	(*-------------------------------------------------------------------------------- Robot Tool Changer Faults -------------------------------------------------------------------*)
	(*Fault1301 - R1 Tool Changer Fault*)
		Fault_Tmrs[1301].PT:= Short_Faults;
		Fault_Tmrs[1301]();
		Fault_Tmrs[1301].IN:= (GTAC_CONFIG.Option_Robot_Count>=1) AND
							MAIN.R1.ToolChanger_FLT;
		Out_To_ICxx.System_Faults[1301]:=Fault_Tmrs[1301].Q;
	(*Fault1302 - R2 Tool Changer Fault*)
		Fault_Tmrs[1302].PT:= Short_Faults;
		Fault_Tmrs[1302]();
		Fault_Tmrs[1302].IN:= (GTAC_CONFIG.Option_Robot_Count>=2) AND
							MAIN.R2.ToolChanger_FLT;
		Out_To_ICxx.System_Faults[1302]:=Fault_Tmrs[1302].Q;
	(*Fault1303 - R3 Tool Changer Fault*)
		Fault_Tmrs[1303].PT:= Short_Faults;
		Fault_Tmrs[1303]();
		Fault_Tmrs[1303].IN:= (GTAC_CONFIG.Option_Robot_Count>=3) AND
							MAIN.R3.ToolChanger_FLT;
		Out_To_ICxx.System_Faults[1303]:=Fault_Tmrs[1303].Q;
	(*Fault1304 - R4 Tool Changer Fault*)
		Fault_Tmrs[1304].PT:= Short_Faults;
		Fault_Tmrs[1304]();
		Fault_Tmrs[1304].IN:= (GTAC_CONFIG.Option_Robot_Count>=4) AND
							MAIN.R4.ToolChanger_FLT;
		Out_To_ICxx.System_Faults[1304]:=Fault_Tmrs[1304].Q;
	(*Fault1305 - R5 Tool Changer Fault*)
		Fault_Tmrs[1305].PT:= Short_Faults;
		Fault_Tmrs[1305]();
		Fault_Tmrs[1305].IN:= (GTAC_CONFIG.Option_Robot_Count>=5) AND
							MAIN.R5.ToolChanger_FLT;
		Out_To_ICxx.System_Faults[1305]:=Fault_Tmrs[1305].Q;
	(*Fault1306 - R6 Tool Changer Fault*)
		Fault_Tmrs[1306].PT:= Short_Faults;
		Fault_Tmrs[1306]();
		Fault_Tmrs[1306].IN:= (GTAC_CONFIG.Option_Robot_Count>=6) AND
							MAIN.R6.ToolChanger_FLT;
		Out_To_ICxx.System_Faults[1306]:=Fault_Tmrs[1306].Q;
	(*Fault1307 - R7 Tool Changer Fault*)
		Fault_Tmrs[1307].PT:= Short_Faults;
		Fault_Tmrs[1307]();
		Fault_Tmrs[1307].IN:= (GTAC_CONFIG.Option_Robot_Count>=7) AND
							MAIN.R7.ToolChanger_FLT;
		Out_To_ICxx.System_Faults[1307]:=Fault_Tmrs[1307].Q;
	(*Fault1308 - R8 Tool Changer Fault*)
		Fault_Tmrs[1308].PT:= Short_Faults;
		Fault_Tmrs[1308]();
		Fault_Tmrs[1308].IN:= (GTAC_CONFIG.Option_Robot_Count>=8) AND
							MAIN.R8.ToolChanger_FLT;
		Out_To_ICxx.System_Faults[1308]:=Fault_Tmrs[1308].Q;
	(*Fault1309 - R9 Tool Changer Fault*)
		Fault_Tmrs[1309].PT:= Short_Faults;
		Fault_Tmrs[1309]();
		Fault_Tmrs[1309].IN:= (GTAC_CONFIG.Option_Robot_Count>=9) AND
							MAIN.R9.ToolChanger_FLT;
		Out_To_ICxx.System_Faults[1309]:=Fault_Tmrs[1309].Q;
	(*Fault1310 - R10 Tool Changer Fault*)
		Fault_Tmrs[1310].PT:= Short_Faults;
		Fault_Tmrs[1310]();
		Fault_Tmrs[1310].IN:= (GTAC_CONFIG.Option_Robot_Count>=10) AND
							MAIN.R10.ToolChanger_FLT;
		Out_To_ICxx.System_Faults[1310]:=Fault_Tmrs[1310].Q;
	(*Fault1311 - R11 Tool Changer Fault*)
		Fault_Tmrs[1311].PT:= Short_Faults;
		Fault_Tmrs[1311]();
		Fault_Tmrs[1311].IN:= (GTAC_CONFIG.Option_Robot_Count>=11) AND
							MAIN.R11.ToolChanger_FLT;
		Out_To_ICxx.System_Faults[1311]:=Fault_Tmrs[1311].Q;
	(*Fault1312 - R12 Tool Changer Fault*)
		Fault_Tmrs[1312].PT:= Short_Faults;
		Fault_Tmrs[1312]();
		Fault_Tmrs[1312].IN:= (GTAC_CONFIG.Option_Robot_Count>=12) AND
							MAIN.R12.ToolChanger_FLT;
		Out_To_ICxx.System_Faults[1312]:=Fault_Tmrs[1312].Q;
	(*Fault1313 - R13 Tool Changer Fault*)
		Fault_Tmrs[1313].PT:= Short_Faults;
		Fault_Tmrs[1313]();
		Fault_Tmrs[1313].IN:= (GTAC_CONFIG.Option_Robot_Count>=13) AND
							MAIN.R13.ToolChanger_FLT;
		Out_To_ICxx.System_Faults[1313]:=Fault_Tmrs[1313].Q;
	(*Fault1314 - R14 Tool Changer Fault*)
		Fault_Tmrs[1314].PT:= Short_Faults;
		Fault_Tmrs[1314]();
		Fault_Tmrs[1314].IN:= (GTAC_CONFIG.Option_Robot_Count>=14) AND
							MAIN.R14.ToolChanger_FLT;
		Out_To_ICxx.System_Faults[1314]:=Fault_Tmrs[1314].Q;
	(*Fault1315 - R15 Tool Changer Fault*)
		Fault_Tmrs[1315].PT:= Short_Faults;
		Fault_Tmrs[1315]();
		Fault_Tmrs[1315].IN:= (GTAC_CONFIG.Option_Robot_Count>=15) AND
							MAIN.R15.ToolChanger_FLT;
		Out_To_ICxx.System_Faults[1315]:=Fault_Tmrs[1315].Q;
	(*Fault1316 - R16 Tool Changer Fault*)
		Fault_Tmrs[1316].PT:= Short_Faults;
		Fault_Tmrs[1316]();
		Fault_Tmrs[1316].IN:= (GTAC_CONFIG.Option_Robot_Count>=16) AND
							MAIN.R16.ToolChanger_FLT;
		Out_To_ICxx.System_Faults[1316]:=Fault_Tmrs[1316].Q;
	(*Fault1317 - R17 Tool Changer Fault*)
		Fault_Tmrs[1317].PT:= Short_Faults;
		Fault_Tmrs[1317]();
		Fault_Tmrs[1317].IN:= (GTAC_CONFIG.Option_Robot_Count>=17) AND
							MAIN.R17.ToolChanger_FLT;
		Out_To_ICxx.System_Faults[1317]:=Fault_Tmrs[1317].Q;
	(*Fault1318 - R18 Tool Changer Fault*)
		Fault_Tmrs[1318].PT:= Short_Faults;
		Fault_Tmrs[1318]();
		Fault_Tmrs[1318].IN:= (GTAC_CONFIG.Option_Robot_Count>=18) AND
							MAIN.R18.ToolChanger_FLT;
		Out_To_ICxx.System_Faults[1318]:=Fault_Tmrs[1318].Q;
	(*Fault1319 - R19 Tool Changer Fault*)
		Fault_Tmrs[1319].PT:= Short_Faults;
		Fault_Tmrs[1319]();
		Fault_Tmrs[1319].IN:= (GTAC_CONFIG.Option_Robot_Count>=19) AND
							MAIN.R19.ToolChanger_FLT;
		Out_To_ICxx.System_Faults[1319]:=Fault_Tmrs[1319].Q;
	(*Fault1320 - R20 Tool Changer Fault*)
		Fault_Tmrs[1320].PT:= Short_Faults;
		Fault_Tmrs[1320]();
		Fault_Tmrs[1320].IN:= (GTAC_CONFIG.Option_Robot_Count>=20) AND
							MAIN.R20.ToolChanger_FLT;
		Out_To_ICxx.System_Faults[1320]:=Fault_Tmrs[1320].Q;
	(*Fault1321 - R21 Tool Changer Fault*)
		Fault_Tmrs[1321].PT:= Short_Faults;
		Fault_Tmrs[1321]();
		Fault_Tmrs[1321].IN:= (GTAC_CONFIG.Option_Robot_Count>=21) AND
							MAIN.R21.ToolChanger_FLT;
		Out_To_ICxx.System_Faults[1321]:=Fault_Tmrs[1321].Q;
	(*Fault1322 - R22 Tool Changer Fault*)
		Fault_Tmrs[1322].PT:= Short_Faults;
		Fault_Tmrs[1322]();
		Fault_Tmrs[1322].IN:= (GTAC_CONFIG.Option_Robot_Count>=22) AND
							MAIN.R22.ToolChanger_FLT;
		Out_To_ICxx.System_Faults[1322]:=Fault_Tmrs[1322].Q;
	(*Fault1323 - R23 Tool Changer Fault*)
		Fault_Tmrs[1323].PT:= Short_Faults;
		Fault_Tmrs[1323]();
		Fault_Tmrs[1323].IN:= (GTAC_CONFIG.Option_Robot_Count>=23) AND
							MAIN.R23.ToolChanger_FLT;
		Out_To_ICxx.System_Faults[1323]:=Fault_Tmrs[1323].Q;
	(*Fault1324 - R24 Tool Changer Fault*)
		Fault_Tmrs[1324].PT:= Short_Faults;
		Fault_Tmrs[1324]();
		Fault_Tmrs[1324].IN:= (GTAC_CONFIG.Option_Robot_Count>=24) AND
							MAIN.R24.ToolChanger_FLT;
		Out_To_ICxx.System_Faults[1324]:=Fault_Tmrs[1324].Q;
	(*Fault1325 - R25 Tool Changer Fault*)
		Fault_Tmrs[1325].PT:= Short_Faults;
		Fault_Tmrs[1325]();
		Fault_Tmrs[1325].IN:= (GTAC_CONFIG.Option_Robot_Count>=25) AND
							MAIN.R25.ToolChanger_FLT;
		Out_To_ICxx.System_Faults[1325]:=Fault_Tmrs[1325].Q;
	(*Fault1326 - R26 Tool Changer Fault*)
		Fault_Tmrs[1326].PT:= Short_Faults;
		Fault_Tmrs[1326]();
		Fault_Tmrs[1326].IN:= (GTAC_CONFIG.Option_Robot_Count>=26) AND
							MAIN.R26.ToolChanger_FLT;
		Out_To_ICxx.System_Faults[1326]:=Fault_Tmrs[1326].Q;
	(*Fault1327 - R27 Tool Changer Fault*)
		Fault_Tmrs[1327].PT:= Short_Faults;
		Fault_Tmrs[1327]();
		Fault_Tmrs[1327].IN:= (GTAC_CONFIG.Option_Robot_Count>=27) AND
							MAIN.R27.ToolChanger_FLT;
		Out_To_ICxx.System_Faults[1327]:=Fault_Tmrs[1327].Q;
	(*Fault1328 - R28 Tool Changer Fault*)
		Fault_Tmrs[1328].PT:= Short_Faults;
		Fault_Tmrs[1328]();
		Fault_Tmrs[1328].IN:= (GTAC_CONFIG.Option_Robot_Count>=28) AND
							MAIN.R28.ToolChanger_FLT;
		Out_To_ICxx.System_Faults[1328]:=Fault_Tmrs[1328].Q;
	(*Fault1329 - R29 Tool Changer Fault*)
		Fault_Tmrs[1329].PT:= Short_Faults;
		Fault_Tmrs[1329]();
		Fault_Tmrs[1329].IN:= (GTAC_CONFIG.Option_Robot_Count>=29) AND
							MAIN.R29.ToolChanger_FLT;
		Out_To_ICxx.System_Faults[1329]:=Fault_Tmrs[1329].Q;
	(*Fault1330 - R30 Tool Changer Fault*)
		Fault_Tmrs[1330].PT:= Short_Faults;
		Fault_Tmrs[1330]();
		Fault_Tmrs[1330].IN:= (GTAC_CONFIG.Option_Robot_Count>=30) AND
							MAIN.R30.ToolChanger_FLT;
		Out_To_ICxx.System_Faults[1330]:=Fault_Tmrs[1330].Q;

	(*-------------------------------------------------------------------------------- Robot EOAT Faults -------------------------------------------------------------------*)
	(*Fault1331 - EOAT01 Fault*)
		Fault_Tmrs[1331].PT:= Short_Faults;
		Fault_Tmrs[1331]();
		Fault_Tmrs[1331].IN:= (MAIN.R1.FB_In.Options.EOAT_Amount>=1) AND
							EOAT01.EOAT_FLT;
		Out_To_ICxx.System_Faults[1331]:=Fault_Tmrs[1331].Q;
	(*Fault1332 - EOAT02 Fault*)
		Fault_Tmrs[1332].PT:= Short_Faults;
		Fault_Tmrs[1332]();
		Fault_Tmrs[1332].IN:= (MAIN.R2.FB_In.Options.EOAT_Amount>=2) AND
							EOAT02.EOAT_FLT;
		Out_To_ICxx.System_Faults[1332]:=Fault_Tmrs[1332].Q;
	(*Fault1333 - EOAT03 Fault*)
		Fault_Tmrs[1333].PT:= Short_Faults;
		Fault_Tmrs[1333]();
		Fault_Tmrs[1333].IN:= (MAIN.R3.FB_In.Options.EOAT_Amount>=3) AND
							EOAT03.EOAT_FLT;
		Out_To_ICxx.System_Faults[1333]:=Fault_Tmrs[1333].Q;
	(*Fault1334 - EOAT04 Fault*)
		Fault_Tmrs[1334].PT:= Short_Faults;
		Fault_Tmrs[1334]();
		Fault_Tmrs[1334].IN:= (MAIN.R4.FB_In.Options.EOAT_Amount>=4) AND
							EOAT04.EOAT_FLT;
		Out_To_ICxx.System_Faults[1334]:=Fault_Tmrs[1334].Q;
	(*Fault1335 - EOAT05 Fault*)
		Fault_Tmrs[1335].PT:= Short_Faults;
		Fault_Tmrs[1335]();
		Fault_Tmrs[1335].IN:= (MAIN.R5.FB_In.Options.EOAT_Amount>=5) AND
							EOAT05.EOAT_FLT;
		Out_To_ICxx.System_Faults[1335]:=Fault_Tmrs[1335].Q;
	(*Fault1336 - EOAT06 Fault*)
		Fault_Tmrs[1336].PT:= Short_Faults;
		Fault_Tmrs[1336]();
		Fault_Tmrs[1336].IN:= (MAIN.R6.FB_In.Options.EOAT_Amount>=6) AND
							EOAT06.EOAT_FLT;
		Out_To_ICxx.System_Faults[1336]:=Fault_Tmrs[1336].Q;
	(*Fault1337 - EOAT07 Fault*)
		Fault_Tmrs[1337].PT:= Short_Faults;
		Fault_Tmrs[1337]();
		Fault_Tmrs[1337].IN:= (MAIN.R7.FB_In.Options.EOAT_Amount>=7) AND
							EOAT07.EOAT_FLT;
		Out_To_ICxx.System_Faults[1337]:=Fault_Tmrs[1337].Q;
	(*Fault1338 - EOAT08 Fault*)
		Fault_Tmrs[1338].PT:= Short_Faults;
		Fault_Tmrs[1338]();
		Fault_Tmrs[1338].IN:= (MAIN.R8.FB_In.Options.EOAT_Amount>=8) AND
							EOAT08.EOAT_FLT;
		Out_To_ICxx.System_Faults[1338]:=Fault_Tmrs[1338].Q;
	(*Fault1339 - EOAT09 Fault*)
		Fault_Tmrs[1339].PT:= Short_Faults;
		Fault_Tmrs[1339]();
		Fault_Tmrs[1339].IN:= (MAIN.R9.FB_In.Options.EOAT_Amount>=9) AND
							EOAT09.EOAT_FLT;
		Out_To_ICxx.System_Faults[1339]:=Fault_Tmrs[1339].Q;
	(*Fault1340 - EOAT10 Fault*)
		Fault_Tmrs[1340].PT:= Short_Faults;
		Fault_Tmrs[1340]();
		Fault_Tmrs[1340].IN:= (MAIN.R10.FB_In.Options.EOAT_Amount>=10) AND
							EOAT10.EOAT_FLT;
		Out_To_ICxx.System_Faults[1340]:=Fault_Tmrs[1340].Q;
(* Note  - add faults as more EOAT are added to the system.
	(*Fault1341 - EOAT11 Fault*)
		Fault_Tmrs[1341].PT:= Short_Faults;
		Fault_Tmrs[1341]();
		Fault_Tmrs[1341].IN:= (GTAC_CONFIG.Option_EOAT_Count>=11) AND
							EOAT11.EOAT_FLT;
		Out_To_ICxx.System_Faults[1341]:=Fault_Tmrs[1341].Q;
	(*Fault1342 - EOAT12 Fault*)
		Fault_Tmrs[1342].PT:= Short_Faults;
		Fault_Tmrs[1342]();
		Fault_Tmrs[1342].IN:= (GTAC_CONFIG.Option_EOAT_Count>=12) AND
							EOAT12.EOAT_FLT;
		Out_To_ICxx.System_Faults[1342]:=Fault_Tmrs[1342].Q;
	(*Fault1343 - EOAT13 Fault*)
		Fault_Tmrs[1343].PT:= Short_Faults;
		Fault_Tmrs[1343]();
		Fault_Tmrs[1343].IN:= (GTAC_CONFIG.Option_EOAT_Count>=13) AND
							EOAT13.EOAT_FLT;
		Out_To_ICxx.System_Faults[1343]:=Fault_Tmrs[1343].Q;
	(*Fault1344 - EOAT14 Fault*)
		Fault_Tmrs[1344].PT:= Short_Faults;
		Fault_Tmrs[1344]();
		Fault_Tmrs[1344].IN:= (GTAC_CONFIG.Option_EOAT_Count>=14) AND
							EOAT14.EOAT_FLT;
		Out_To_ICxx.System_Faults[1344]:=Fault_Tmrs[1344].Q;
	(*Fault1345 - EOAT15 Fault*)
		Fault_Tmrs[1345].PT:= Short_Faults;
		Fault_Tmrs[1345]();
		Fault_Tmrs[1345].IN:= (GTAC_CONFIG.Option_EOAT_Count>=15) AND
							EOAT15.EOAT_FLT;
		Out_To_ICxx.System_Faults[1345]:=Fault_Tmrs[1345].Q;
	(*Fault1346 - EOAT16 Fault*)
		Fault_Tmrs[1346].PT:= Short_Faults;
		Fault_Tmrs[1346]();
		Fault_Tmrs[1346].IN:= (GTAC_CONFIG.Option_EOAT_Count>=16) AND
							EOAT16.EOAT_FLT;
		Out_To_ICxx.System_Faults[1346]:=Fault_Tmrs[1346].Q;
	(*Fault1347 - EOAT17 Fault*)
		Fault_Tmrs[1347].PT:= Short_Faults;
		Fault_Tmrs[1347]();
		Fault_Tmrs[1347].IN:= (GTAC_CONFIG.Option_EOAT_Count>=17) AND
							EOAT17.EOAT_FLT;
		Out_To_ICxx.System_Faults[1347]:=Fault_Tmrs[1347].Q;
	(*Fault1348 - EOAT18 Fault*)
		Fault_Tmrs[1348].PT:= Short_Faults;
		Fault_Tmrs[1348]();
		Fault_Tmrs[1348].IN:= (GTAC_CONFIG.Option_EOAT_Count>=18) AND
							EOAT18.EOAT_FLT;
		Out_To_ICxx.System_Faults[1348]:=Fault_Tmrs[1348].Q;
	(*Fault1349 - EOAT19 Fault*)
		Fault_Tmrs[1349].PT:= Short_Faults;
		Fault_Tmrs[1349]();
		Fault_Tmrs[1349].IN:= (GTAC_CONFIG.Option_EOAT_Count>=19) AND
							EOAT19.EOAT_FLT;
		Out_To_ICxx.System_Faults[1349]:=Fault_Tmrs[1349].Q;
	(*Fault1350 - EOAT20 Fault*)
		Fault_Tmrs[1350].PT:= Short_Faults;
		Fault_Tmrs[1350]();
		Fault_Tmrs[1350].IN:= (GTAC_CONFIG.Option_EOAT_Count>=20) AND
							EOAT20.EOAT_FLT;
		Out_To_ICxx.System_Faults[1350]:=Fault_Tmrs[1350].Q;
	(*Fault1351 - EOAT21 Fault*)
		Fault_Tmrs[1351].PT:= Short_Faults;
		Fault_Tmrs[1351]();
		Fault_Tmrs[1351].IN:= (GTAC_CONFIG.Option_EOAT_Count>=21) AND
							EOAT21.EOAT_FLT;
		Out_To_ICxx.System_Faults[1351]:=Fault_Tmrs[1351].Q;
	(*Fault1352 - EOAT22 Fault*)
		Fault_Tmrs[1352].PT:= Short_Faults;
		Fault_Tmrs[1352]();
		Fault_Tmrs[1352].IN:= (GTAC_CONFIG.Option_EOAT_Count>=22) AND
							EOAT22.EOAT_FLT;
		Out_To_ICxx.System_Faults[1352]:=Fault_Tmrs[1352].Q;
	(*Fault1353 - EOAT23 Fault*)
		Fault_Tmrs[1353].PT:= Short_Faults;
		Fault_Tmrs[1353]();
		Fault_Tmrs[1353].IN:= (GTAC_CONFIG.Option_EOAT_Count>=23) AND
							EOAT23.EOAT_FLT;
		Out_To_ICxx.System_Faults[1353]:=Fault_Tmrs[1353].Q;
	(*Fault1354 - EOAT24 Fault*)
		Fault_Tmrs[1354].PT:= Short_Faults;
		Fault_Tmrs[1354]();
		Fault_Tmrs[1354].IN:= (GTAC_CONFIG.Option_EOAT_Count>=24) AND
							EOAT24.EOAT_FLT;
		Out_To_ICxx.System_Faults[1354]:=Fault_Tmrs[1354].Q;
	(*Fault1355 - EOAT25 Fault*)
		Fault_Tmrs[1355].PT:= Short_Faults;
		Fault_Tmrs[1355]();
		Fault_Tmrs[1355].IN:= (GTAC_CONFIG.Option_EOAT_Count>=25) AND
							EOAT25.EOAT_FLT;
		Out_To_ICxx.System_Faults[1355]:=Fault_Tmrs[1355].Q;
	(*Fault1356 - EOAT26 Fault*)
		Fault_Tmrs[1356].PT:= Short_Faults;
		Fault_Tmrs[1356]();
		Fault_Tmrs[1356].IN:= (GTAC_CONFIG.Option_EOAT_Count>=26) AND
							EOAT26.EOAT_FLT;
		Out_To_ICxx.System_Faults[1356]:=Fault_Tmrs[1356].Q;
	(*Fault1357 - EOAT27 Fault*)
		Fault_Tmrs[1357].PT:= Short_Faults;
		Fault_Tmrs[1357]();
		Fault_Tmrs[1357].IN:= (GTAC_CONFIG.Option_EOAT_Count>=27) AND
							EOAT27.EOAT_FLT;
		Out_To_ICxx.System_Faults[1357]:=Fault_Tmrs[1357].Q;
	(*Fault1358 - EOAT28 Fault*)
		Fault_Tmrs[1358].PT:= Short_Faults;
		Fault_Tmrs[1358]();
		Fault_Tmrs[1358].IN:= (GTAC_CONFIG.Option_EOAT_Count>=28) AND
							EOAT28.EOAT_FLT;
		Out_To_ICxx.System_Faults[1358]:=Fault_Tmrs[1358].Q;
	(*Fault1359 - EOAT29 Fault*)
		Fault_Tmrs[1359].PT:= Short_Faults;
		Fault_Tmrs[1359]();
		Fault_Tmrs[1359].IN:= (GTAC_CONFIG.Option_EOAT_Count>=29) AND
							EOAT29.EOAT_FLT;
		Out_To_ICxx.System_Faults[1359]:=Fault_Tmrs[1359].Q;
	(*Fault1360 - EOAT30 Fault*)
		Fault_Tmrs[1360].PT:= Short_Faults;
		Fault_Tmrs[1360]();
		Fault_Tmrs[1360].IN:= (GTAC_CONFIG.Option_EOAT_Count>=30) AND
							EOAT30.EOAT_FLT;
		Out_To_ICxx.System_Faults[1360]:=Fault_Tmrs[1360].Q;*)
	(*--------------------------------------------------------------------------------  TurnTable Positioning Faults -------------------------------------------------------------------*)
	(*DEBUG, add Turn / DialTable Positioning / Switch Faults here, as required*)

	(*Fault1421 - TT01 Positioning / Switch Fault*)
		Fault_Tmrs[1421].PT:= Short_Faults;
		Fault_Tmrs[1421]();
		Fault_Tmrs[1421].IN:= FALSE;
		Out_To_ICxx.System_Faults[1421]:=Fault_Tmrs[1421].Q;
	(*Fault1422 - TT02 Positioning / Switch Fault*)
		Fault_Tmrs[1422].PT:= Short_Faults;
		Fault_Tmrs[1422]();
		Fault_Tmrs[1422].IN:= FALSE;
		Out_To_ICxx.System_Faults[1422]:=Fault_Tmrs[1422].Q;
	(*Fault1423 - TT03 Positioning / Switch Fault*)
		Fault_Tmrs[1423].PT:= Short_Faults;
		Fault_Tmrs[1423]();
		Fault_Tmrs[1423].IN:= FALSE;
		Out_To_ICxx.System_Faults[1423]:=Fault_Tmrs[1423].Q;
	(*Fault1424 - TT04 Positioning / Switch Fault*)
		Fault_Tmrs[1424].PT:= Short_Faults;
		Fault_Tmrs[1424]();
		Fault_Tmrs[1424].IN:= FALSE;
		Out_To_ICxx.System_Faults[1424]:=Fault_Tmrs[1424].Q;
	(*Fault1425 - TT05 Positioning / Switch Fault*)
		Fault_Tmrs[1425].PT:= Short_Faults;
		Fault_Tmrs[1425]();
		Fault_Tmrs[1425].IN:= FALSE;
		Out_To_ICxx.System_Faults[1425]:=Fault_Tmrs[1425].Q;
	(*Fault1426 - TT06 Positioning / Switch  Fault*)
		Fault_Tmrs[1426].PT:= Short_Faults;
		Fault_Tmrs[1426]();
		Fault_Tmrs[1426].IN:= FALSE;
		Out_To_ICxx.System_Faults[1426]:=Fault_Tmrs[1426].Q;
	(*Fault1427 - TT07 Positioning / Switch Fault*)
		Fault_Tmrs[1427].PT:= Short_Faults;
		Fault_Tmrs[1427]();
		Fault_Tmrs[1427].IN:= FALSE;
		Out_To_ICxx.System_Faults[1427]:=Fault_Tmrs[1427].Q;
	(*Fault1428 - TT08 Positioning / Switch Fault*)
		Fault_Tmrs[1428].PT:= Short_Faults;
		Fault_Tmrs[1428]();
		Fault_Tmrs[1428].IN:= FALSE;
		Out_To_ICxx.System_Faults[1428]:=Fault_Tmrs[1428].Q;
	(*Fault1299 - TT09 Positioning / Switch Fault*)
		Fault_Tmrs[1429].PT:= Short_Faults;
		Fault_Tmrs[1429]();
		Fault_Tmrs[1429].IN:= FALSE;
		Out_To_ICxx.System_Faults[1429]:=Fault_Tmrs[1429].Q;

	(*--------------------------------------------------------------------------------  Pedestal Station Faults -------------------------------------------------------------------*)
	(*Fault1431 - Ped01 Fault*)
		Fault_Tmrs[1431].PT:= Short_Faults;
		Fault_Tmrs[1431]();
		Fault_Tmrs[1431].IN:= (GTAC_CONFIG.Option_Ped_Count>=1) AND
							((MAIN.Ped[1].CLFaulted<>0) OR (MAIN.Ped[1].PPFaulted<>0) OR NOT Main.Ped[1].DiscreteNode_OK);
		Out_To_ICxx.System_Faults[1431]:=Fault_Tmrs[1431].Q;
	(*Fault1432 - Ped02 Fault*)
		Fault_Tmrs[1432].PT:= Short_Faults;
		Fault_Tmrs[1432]();
		Fault_Tmrs[1432].IN:= (GTAC_CONFIG.Option_Ped_Count>=2) AND
							((MAIN.Ped[2].CLFaulted<>0) OR (MAIN.Ped[2].PPFaulted<>0) OR NOT Main.Ped[2].DiscreteNode_OK);
		Out_To_ICxx.System_Faults[1432]:=Fault_Tmrs[1432].Q;
	(*Fault1433 - Ped03 Fault*)
		Fault_Tmrs[1433].PT:= Short_Faults;
		Fault_Tmrs[1433]();
		Fault_Tmrs[1433].IN:= (GTAC_CONFIG.Option_Ped_Count>=3) AND
							((MAIN.Ped[3].CLFaulted<>0) OR (MAIN.Ped[3].PPFaulted<>0) OR NOT Main.Ped[3].DiscreteNode_OK);
		Out_To_ICxx.System_Faults[1433]:=Fault_Tmrs[1433].Q;
	(*Fault1434 - Ped4 Fault*)
		Fault_Tmrs[1434].PT:= Short_Faults;
		Fault_Tmrs[1434]();
		Fault_Tmrs[1434].IN:= (GTAC_CONFIG.Option_Ped_Count>=4) AND
							((MAIN.Ped[4].CLFaulted<>0) OR (MAIN.Ped[4].PPFaulted<>0) OR NOT Main.Ped[4].DiscreteNode_OK);
		Out_To_ICxx.System_Faults[1434]:=Fault_Tmrs[1434].Q;
	(*Fault1435 - Ped5 Fault*)
		Fault_Tmrs[1435].PT:= Short_Faults;
		Fault_Tmrs[1435]();
		Fault_Tmrs[1435].IN:= (GTAC_CONFIG.Option_Ped_Count>=5) AND
							((MAIN.Ped[5].CLFaulted<>0) OR (MAIN.Ped[5].PPFaulted<>0) OR NOT Main.Ped[5].DiscreteNode_OK);
		Out_To_ICxx.System_Faults[1435]:=Fault_Tmrs[1435].Q;
	(*Fault1436 - Ped6 Fault*)
		Fault_Tmrs[1436].PT:= Short_Faults;
		Fault_Tmrs[1436]();
		Fault_Tmrs[1436].IN:= (GTAC_CONFIG.Option_Ped_Count>=6) AND
							((MAIN.Ped[6].CLFaulted<>0) OR (MAIN.Ped[6].PPFaulted<>0) OR NOT Main.Ped[6].DiscreteNode_OK);
		Out_To_ICxx.System_Faults[1436]:=Fault_Tmrs[1436].Q;
	(*Fault1437 - Ped7 Fault*)
		Fault_Tmrs[1437].PT:= Short_Faults;
		Fault_Tmrs[1437]();
		Fault_Tmrs[1437].IN:= (GTAC_CONFIG.Option_Ped_Count>=7) AND
							((MAIN.Ped[7].CLFaulted<>0) OR (MAIN.Ped[7].PPFaulted<>0) OR NOT Main.Ped[7].DiscreteNode_OK);
		Out_To_ICxx.System_Faults[1437]:=Fault_Tmrs[1437].Q;
	(*Fault1438 - Ped8 Fault*)
		Fault_Tmrs[1438].PT:= Short_Faults;
		Fault_Tmrs[1438]();
		Fault_Tmrs[1438].IN:= (GTAC_CONFIG.Option_Ped_Count>=8) AND
							((MAIN.Ped[8].CLFaulted<>0) OR (MAIN.Ped[8].PPFaulted<>0) OR NOT Main.Ped[8].DiscreteNode_OK);
		Out_To_ICxx.System_Faults[1438]:=Fault_Tmrs[1438].Q;
	(*Fault1439 - Ped9 Fault*)
		Fault_Tmrs[1439].PT:= Short_Faults;
		Fault_Tmrs[1439]();
		Fault_Tmrs[1439].IN:= (GTAC_CONFIG.Option_Ped_Count>=9) AND
							((MAIN.Ped[9].CLFaulted<>0) OR (MAIN.Ped[9].PPFaulted<>0) OR NOT Main.Ped[9].DiscreteNode_OK);
		Out_To_ICxx.System_Faults[1439]:=Fault_Tmrs[1439].Q;
	(*Fault1440 - Ped10 Fault*)
		Fault_Tmrs[1440].PT:= Short_Faults;
		Fault_Tmrs[1440]();
		Fault_Tmrs[1440].IN:= (GTAC_CONFIG.Option_Ped_Count>=10) AND
							((MAIN.Ped[10].CLFaulted<>0) OR (MAIN.Ped[10].PPFaulted<>0) OR NOT Main.Ped[10].DiscreteNode_OK);
		Out_To_ICxx.System_Faults[1440]:=Fault_Tmrs[1440].Q;
	(*Fault1441 - Ped11 Fault*)
		Fault_Tmrs[1441].PT:= Short_Faults;
		Fault_Tmrs[1441]();
		Fault_Tmrs[1441].IN:= (GTAC_CONFIG.Option_Ped_Count>=11) AND
							((MAIN.Ped[11].CLFaulted<>0) OR (MAIN.Ped[11].PPFaulted<>0) OR NOT Main.Ped[11].DiscreteNode_OK);
		Out_To_ICxx.System_Faults[1441]:=Fault_Tmrs[1441].Q;
	(*Fault1442 - Ped12 Fault*)
		Fault_Tmrs[1442].PT:= Short_Faults;
		Fault_Tmrs[1442]();
		Fault_Tmrs[1442].IN:= (GTAC_CONFIG.Option_Ped_Count>=12) AND
							((MAIN.Ped[12].CLFaulted<>0) OR (MAIN.Ped[12].PPFaulted<>0) OR NOT Main.Ped[12].DiscreteNode_OK);
		Out_To_ICxx.System_Faults[1442]:=Fault_Tmrs[1442].Q;
	(*Fault1443 - Ped13 Fault*)
		Fault_Tmrs[1443].PT:= Short_Faults;
		Fault_Tmrs[1443]();
		Fault_Tmrs[1443].IN:= (GTAC_CONFIG.Option_Ped_Count>=13) AND
							((MAIN.Ped[13].CLFaulted<>0) OR (MAIN.Ped[13].PPFaulted<>0) OR NOT Main.Ped[13].DiscreteNode_OK);
		Out_To_ICxx.System_Faults[1443]:=Fault_Tmrs[1443].Q;
	(*Fault1444 - Ped14 Fault*)
		Fault_Tmrs[1444].PT:= Short_Faults;
		Fault_Tmrs[1444]();
		Fault_Tmrs[1444].IN:= (GTAC_CONFIG.Option_Ped_Count>=14) AND
							((MAIN.Ped[14].CLFaulted<>0) OR (MAIN.Ped[14].PPFaulted<>0) OR NOT Main.Ped[14].DiscreteNode_OK);
		Out_To_ICxx.System_Faults[1444]:=Fault_Tmrs[1444].Q;
	(*Fault1445 - Ped15 Fault*)
		Fault_Tmrs[1445].PT:= Short_Faults;
		Fault_Tmrs[1445]();
		Fault_Tmrs[1445].IN:= (GTAC_CONFIG.Option_Ped_Count>=15) AND
							((MAIN.Ped[15].CLFaulted<>0) OR (MAIN.Ped[15].PPFaulted<>0) OR NOT Main.Ped[15].DiscreteNode_OK);
		Out_To_ICxx.System_Faults[1445]:=Fault_Tmrs[1445].Q;
	(*Fault1446 - Ped16 Fault*)
		Fault_Tmrs[1446].PT:= Short_Faults;
		Fault_Tmrs[1446]();
		Fault_Tmrs[1446].IN:= (GTAC_CONFIG.Option_Ped_Count>=16) AND
							((MAIN.Ped[16].CLFaulted<>0) OR (MAIN.Ped[16].PPFaulted<>0) OR NOT Main.Ped[16].DiscreteNode_OK);
		Out_To_ICxx.System_Faults[1446]:=Fault_Tmrs[1446].Q;
	(*Fault1447 - Ped17 Fault*)
		Fault_Tmrs[1447].PT:= Short_Faults;
		Fault_Tmrs[1447]();
		Fault_Tmrs[1447].IN:= (GTAC_CONFIG.Option_Ped_Count>=17) AND
							((MAIN.Ped[17].CLFaulted<>0) OR (MAIN.Ped[17].PPFaulted<>0) OR NOT Main.Ped[17].DiscreteNode_OK);
		Out_To_ICxx.System_Faults[1447]:=Fault_Tmrs[1447].Q;
	(*Fault1448 - Ped18 Fault*)
		Fault_Tmrs[1448].PT:= Short_Faults;
		Fault_Tmrs[1448]();
		Fault_Tmrs[1448].IN:= (GTAC_CONFIG.Option_Ped_Count>=18) AND
							((MAIN.Ped[18].CLFaulted<>0) OR (MAIN.Ped[18].PPFaulted<>0) OR NOT Main.Ped[18].DiscreteNode_OK);
		Out_To_ICxx.System_Faults[1448]:=Fault_Tmrs[1448].Q;
	(*Fault1449 - Ped19 Fault*)
		Fault_Tmrs[1449].PT:= Short_Faults;
		Fault_Tmrs[1449]();
		Fault_Tmrs[1449].IN:= (GTAC_CONFIG.Option_Ped_Count>=19) AND
							((MAIN.Ped[19].CLFaulted<>0) OR (MAIN.Ped[19].PPFaulted<>0) OR NOT Main.Ped[19].DiscreteNode_OK);
		Out_To_ICxx.System_Faults[1449]:=Fault_Tmrs[1449].Q;
	(*Fault1450 - Ped20 Fault*)
		Fault_Tmrs[1450].PT:= Short_Faults;
		Fault_Tmrs[1450]();
		Fault_Tmrs[1450].IN:= (GTAC_CONFIG.Option_Ped_Count>=20) AND
							((MAIN.Ped[20].CLFaulted<>0) OR (MAIN.Ped[20].PPFaulted<>0) OR NOT Main.Ped[20].DiscreteNode_OK);
		Out_To_ICxx.System_Faults[1450]:=Fault_Tmrs[1450].Q;
	(*Fault1451 - Ped21 Fault*)
		Fault_Tmrs[1451].PT:= Short_Faults;
		Fault_Tmrs[1451]();
		Fault_Tmrs[1451].IN:= (GTAC_CONFIG.Option_Ped_Count>=21) AND
							((MAIN.Ped[21].CLFaulted<>0) OR (MAIN.Ped[21].PPFaulted<>0) OR NOT Main.Ped[21].DiscreteNode_OK);
		Out_To_ICxx.System_Faults[1451]:=Fault_Tmrs[1451].Q;
	(*Fault1452 - Ped22 Fault*)
		Fault_Tmrs[1452].PT:= Short_Faults;
		Fault_Tmrs[1452]();
		Fault_Tmrs[1452].IN:= (GTAC_CONFIG.Option_Ped_Count>=22) AND
							((MAIN.Ped[22].CLFaulted<>0) OR (MAIN.Ped[22].PPFaulted<>0) OR NOT Main.Ped[22].DiscreteNode_OK);
		Out_To_ICxx.System_Faults[1452]:=Fault_Tmrs[1452].Q;
	(*Fault1453 - Ped23 Fault*)
		Fault_Tmrs[1453].PT:= Short_Faults;
		Fault_Tmrs[1453]();
		Fault_Tmrs[1453].IN:= (GTAC_CONFIG.Option_Ped_Count>=23) AND
							((MAIN.Ped[23].CLFaulted<>0) OR (MAIN.Ped[23].PPFaulted<>0) OR NOT Main.Ped[23].DiscreteNode_OK);
		Out_To_ICxx.System_Faults[1453]:=Fault_Tmrs[1453].Q;
	(*Fault1454 - Ped24 Fault*)
		Fault_Tmrs[1454].PT:= Short_Faults;
		Fault_Tmrs[1454]();
		Fault_Tmrs[1454].IN:= (GTAC_CONFIG.Option_Ped_Count>=24) AND
							((MAIN.Ped[24].CLFaulted<>0) OR (MAIN.Ped[24].PPFaulted<>0) OR NOT Main.Ped[24].DiscreteNode_OK);
		Out_To_ICxx.System_Faults[1454]:=Fault_Tmrs[1454].Q;
	(*Fault1455 - Ped25 Fault*)
		Fault_Tmrs[1455].PT:= Short_Faults;
		Fault_Tmrs[1455]();
		Fault_Tmrs[1455].IN:= (GTAC_CONFIG.Option_Ped_Count>=25) AND
							((MAIN.Ped[25].CLFaulted<>0) OR (MAIN.Ped[25].PPFaulted<>0) OR NOT Main.Ped[25].DiscreteNode_OK);
		Out_To_ICxx.System_Faults[1455]:=Fault_Tmrs[1455].Q;
	(*Fault1456 - Ped26 Fault*)
		Fault_Tmrs[1456].PT:= Short_Faults;
		Fault_Tmrs[1456]();
		Fault_Tmrs[1456].IN:= (GTAC_CONFIG.Option_Ped_Count>=26) AND
							((MAIN.Ped[26].CLFaulted<>0) OR (MAIN.Ped[26].PPFaulted<>0) OR NOT Main.Ped[26].DiscreteNode_OK);
		Out_To_ICxx.System_Faults[1456]:=Fault_Tmrs[1456].Q;
	(*Fault1457 - Ped27 Fault*)
		Fault_Tmrs[1457].PT:= Short_Faults;
		Fault_Tmrs[1457]();
		Fault_Tmrs[1457].IN:= (GTAC_CONFIG.Option_Ped_Count>=27) AND
							((MAIN.Ped[27].CLFaulted<>0) OR (MAIN.Ped[27].PPFaulted<>0) OR NOT Main.Ped[27].DiscreteNode_OK);
		Out_To_ICxx.System_Faults[1457]:=Fault_Tmrs[1457].Q;
	(*Fault1458 - Ped28 Fault*)
		Fault_Tmrs[1458].PT:= Short_Faults;
		Fault_Tmrs[1458]();
		Fault_Tmrs[1458].IN:= (GTAC_CONFIG.Option_Ped_Count>=28) AND
							((MAIN.Ped[28].CLFaulted<>0) OR (MAIN.Ped[28].PPFaulted<>0) OR NOT Main.Ped[28].DiscreteNode_OK);
		Out_To_ICxx.System_Faults[1458]:=Fault_Tmrs[1458].Q;
	(*Fault1459 - Ped29 Fault*)
		Fault_Tmrs[1459].PT:= Short_Faults;
		Fault_Tmrs[1459]();
		Fault_Tmrs[1459].IN:= (GTAC_CONFIG.Option_Ped_Count>=29) AND
							((MAIN.Ped[29].CLFaulted<>0) OR (MAIN.Ped[29].PPFaulted<>0) OR NOT Main.Ped[29].DiscreteNode_OK);
		Out_To_ICxx.System_Faults[1459]:=Fault_Tmrs[1459].Q;
	(*Fault1460 - Ped30 Fault*)
		Fault_Tmrs[1460].PT:= Short_Faults;
		Fault_Tmrs[1460]();
		Fault_Tmrs[1460].IN:= (GTAC_CONFIG.Option_Ped_Count>=30) AND
							((MAIN.Ped[30].CLFaulted<>0) OR (MAIN.Ped[30].PPFaulted<>0) OR NOT Main.Ped[30].DiscreteNode_OK);
		Out_To_ICxx.System_Faults[1460]:=Fault_Tmrs[1460].Q;


	(*--------------------------------------------------------------------- Stud Controller Faults ------------------------------------------------------*)

	(*Fault1465 - Stud Controller1 Fault*)
		Fault_Tmrs[1465].PT:= Long_Faults;
		Fault_Tmrs[1465]();
		Fault_Tmrs[1465].IN:= (GTAC_CONFIG.Option_StudController_Count>=1) AND
							 MAIN.ST01.Faulted ;
		Out_To_ICxx.System_Faults[1465]:=Fault_Tmrs[1465].Q;
	(*Fault1466 - Stud Controller2 Fault*)
		Fault_Tmrs[1466].PT:= Long_Faults;
		Fault_Tmrs[1466]();
		Fault_Tmrs[1466].IN:= (GTAC_CONFIG.Option_StudController_Count>=2) AND
							MAIN.ST02.Faulted ;
		Out_To_ICxx.System_Faults[1466]:=Fault_Tmrs[1466].Q;
	(*Fault1467 - Stud Controller3 Fault*)
		Fault_Tmrs[1467].PT:= Long_Faults;
		Fault_Tmrs[1467]();
		Fault_Tmrs[1467].IN:= (GTAC_CONFIG.Option_StudController_Count>=3) AND
							MAIN.ST03.Faulted ;
		Out_To_ICxx.System_Faults[1467]:=Fault_Tmrs[1467].Q;
	(*Fault1468 - Stud Controller4 Fault*)
		Fault_Tmrs[1468].PT:= Long_Faults;
		Fault_Tmrs[1468]();
		Fault_Tmrs[1468].IN:= (GTAC_CONFIG.Option_StudController_Count>=1) AND
							MAIN.ST04.Faulted ;
		Out_To_ICxx.System_Faults[1468]:=Fault_Tmrs[1468].Q;
	(*Fault1469 - Stud Controller5 Fault*)
		Fault_Tmrs[1469].PT:= Long_Faults;
		Fault_Tmrs[1469]();
		Fault_Tmrs[1469].IN:= FALSE;
		Out_To_ICxx.System_Faults[1469]:=Fault_Tmrs[1469].Q;
	(*Fault1470 - Stud Controller6 Fault*)
		Fault_Tmrs[1470].PT:= Long_Faults;
		Fault_Tmrs[1470]();
		Fault_Tmrs[1470].IN:= FALSE;
		Out_To_ICxx.System_Faults[1470]:=Fault_Tmrs[1470].Q;
	(*Fault1471 - Stud Controller7 Fault*)
		Fault_Tmrs[1471].PT:= Long_Faults;
		Fault_Tmrs[1471]();
		Fault_Tmrs[1471].IN:= FALSE;
		Out_To_ICxx.System_Faults[1471]:=Fault_Tmrs[1471].Q;
	(*Fault1472 - Stud Controller8 Fault*)
		Fault_Tmrs[1472].PT:= Long_Faults;
		Fault_Tmrs[1472]();
		Fault_Tmrs[1472].IN:= FALSE;
		Out_To_ICxx.System_Faults[1472]:=Fault_Tmrs[1472].Q;
	(*Fault1473 - Stud Controller9 Fault*)
		Fault_Tmrs[1473].PT:= Long_Faults;
		Fault_Tmrs[1473]();
		Fault_Tmrs[1473].IN:= FALSE;
		Out_To_ICxx.System_Faults[1473]:=Fault_Tmrs[1473].Q;

	(*--------------------------------------------------------------------- Sealant Controller Faults ------------------------------------------------------*)
	
	(*Fault1475 - Sealant Controller1 Fault*)
		Fault_Tmrs[1475].PT:= Short_Faults;
		Fault_Tmrs[1475]();
		Fault_Tmrs[1475].IN:= (GTAC_CONFIG.Option_SealController_Count>=1) AND
							MAIN.SL01.Faulted;
		Out_To_ICxx.System_Faults[1475]:=Fault_Tmrs[1475].Q;
	(*Fault1476 - Sealant Controller2 Fault*)
		Fault_Tmrs[1476].PT:= Short_Faults;
		Fault_Tmrs[1476]();
		Fault_Tmrs[1476].IN:= (GTAC_CONFIG.Option_SealController_Count>=2) AND
							MAIN.SL02.Faulted;
		Out_To_ICxx.System_Faults[1476]:=Fault_Tmrs[1476].Q;
	(*Fault1477 - Sealant Controller3 Fault*)
		Fault_Tmrs[1477].PT:= Short_Faults;
		Fault_Tmrs[1477]();
		Fault_Tmrs[1477].IN:= (GTAC_CONFIG.Option_SealController_Count>=3) AND
							MAIN.SL03.Faulted;
		Out_To_ICxx.System_Faults[1477]:=Fault_Tmrs[1477].Q;
	(*Fault1478 - Sealant Controller4 Fault*)
		Fault_Tmrs[1478].PT:= Short_Faults;
		Fault_Tmrs[1478]();
		Fault_Tmrs[1478].IN:= (GTAC_CONFIG.Option_SealController_Count>=4) AND
							MAIN.SL04.Faulted;
		Out_To_ICxx.System_Faults[1478]:=Fault_Tmrs[1478].Q;
	(*Fault1479 - Sealant Controller5 Fault*)
		Fault_Tmrs[1479].PT:= Short_Faults;
		Fault_Tmrs[1479]();
		Fault_Tmrs[1479].IN:= FALSE;
		Out_To_ICxx.System_Faults[1479]:=Fault_Tmrs[1479].Q;
	(*Fault1480 - Sealant Controller6 Fault*)
		Fault_Tmrs[1480].PT:= Short_Faults;
		Fault_Tmrs[1480]();
		Fault_Tmrs[1480].IN:= FALSE;
		Out_To_ICxx.System_Faults[1480]:=Fault_Tmrs[1480].Q;
	(*Fault1481 - Sealant Controller7 Fault*)
		Fault_Tmrs[1481].PT:= Short_Faults;
		Fault_Tmrs[1481]();
		Fault_Tmrs[1481].IN:= FALSE;
		Out_To_ICxx.System_Faults[1481]:=Fault_Tmrs[1481].Q;
	(*Fault1482 - Sealant Controller8 Fault*)
		Fault_Tmrs[1482].PT:= Short_Faults;
		Fault_Tmrs[1482]();
		Fault_Tmrs[1482].IN:= FALSE;
		Out_To_ICxx.System_Faults[1482]:=Fault_Tmrs[1482].Q;
	(*Fault1483 - Sealant Controller9 Fault*)
		Fault_Tmrs[1483].PT:= Short_Faults;
		Fault_Tmrs[1483]();
		Fault_Tmrs[1483].IN:= FALSE;
		Out_To_ICxx.System_Faults[1483]:=Fault_Tmrs[1483].Q;

	(*--------------------------------------------------------------------- Nut Weld System Faults ------------------------------------------------------*)
	(*Add as required
	(*Fault1485 - Nut Welder1 Fault*)
		Fault_Tmrs[1485].PT:= Short_Faults;
		Fault_Tmrs[1485]();
		Fault_Tmrs[1485].IN:= (NW01.CLFaults<>0) OR (NW01.PPFaults<>0);
		Out_To_ICxx.System_Faults[1485]:=Fault_Tmrs[1485].Q;
	(*Fault1486 - Nut Welder2 Fault*)
		Fault_Tmrs[1486].PT:= Short_Faults;
		Fault_Tmrs[1486]();
		Fault_Tmrs[1486].IN:= (NW02.CLFaults<>0) OR (NW02.PPFaults<>0);
		Out_To_ICxx.System_Faults[1486]:=Fault_Tmrs[1486].Q;
	(*Fault1487 - Nut Welder3 Fault*)
		Fault_Tmrs[1487].PT:= Short_Faults;
		Fault_Tmrs[1487]();
		Fault_Tmrs[1487].IN:= (NW03.CLFaults<>0) OR (NW03.PPFaults<>0);
		Out_To_ICxx.System_Faults[1487]:=Fault_Tmrs[1487].Q;
	(*Fault1488 - Nut Welder4 Fault*)
		Fault_Tmrs[1488].PT:= Short_Faults;
		Fault_Tmrs[1488]();
		Fault_Tmrs[1488].IN:= (NW04.CLFaults<>0) OR (NW04.PPFaults<>0);
		Out_To_ICxx.System_Faults[1488]:=Fault_Tmrs[1488].Q;
	(*Fault1489 - Nut Welder5 Fault*)
		Fault_Tmrs[1489].PT:= Short_Faults;
		Fault_Tmrs[1489]();
		Fault_Tmrs[1489].IN:= (NW05.CLFaults<>0) OR (NW05.PPFaults<>0);
		Out_To_ICxx.System_Faults[1489]:=Fault_Tmrs[1489].Q;
	*)
	(* ---------------------------------------------------------------------------- MD Door Faults -----------------------------------------------------------------------------------------*)
	
	(*Fault1491 - MD01 Door Faulted*)
		Fault_Tmrs[1491].PT:= Short_Faults;
		Fault_Tmrs[1491]();
		Fault_Tmrs[1491].IN:= (GTAC_CONFIG.Option_MD_Count>=1) AND
							MAIN.MD01.Door_Faulted;
		Out_To_ICxx.System_Faults[1491]:=Fault_Tmrs[1491].Q;
	(*Fault1492 - MD02 Door Faulted*)
		Fault_Tmrs[1492].PT:= Short_Faults;
		Fault_Tmrs[1492]();
		Fault_Tmrs[1492].IN:= (GTAC_CONFIG.Option_MD_Count>=2) AND
							MAIN.MD02.Door_Faulted;
		Out_To_ICxx.System_Faults[1492]:=Fault_Tmrs[1492].Q;
	(*Fault1493 - MD03 Door Faulted*)
		Fault_Tmrs[1493].PT:= Short_Faults;
		Fault_Tmrs[1493]();
		Fault_Tmrs[1493].IN:= (GTAC_CONFIG.Option_MD_Count>=3) AND
							MAIN.MD03.Door_Faulted;
		Out_To_ICxx.System_Faults[1493]:=Fault_Tmrs[1493].Q;
	(*Fault1494 - MD04 Door Faulted*)
		Fault_Tmrs[1494].PT:= Short_Faults;
		Fault_Tmrs[1494]();
		Fault_Tmrs[1494].IN:= (GTAC_CONFIG.Option_MD_Count>=4) AND
							MAIN.MD04.Door_Faulted;
		Out_To_ICxx.System_Faults[1494]:=Fault_Tmrs[1494].Q;
	(*Fault1495 - MD05 Door Faulted*)
		Fault_Tmrs[1495].PT:= Short_Faults;
		Fault_Tmrs[1495]();
		Fault_Tmrs[1495].IN:= (GTAC_CONFIG.Option_MD_Count>=5) AND
							MAIN.MD05.Door_Faulted;
		Out_To_ICxx.System_Faults[1495]:=Fault_Tmrs[1495].Q;


	(* ---------------------------------------------------------------------------- VFD General Faults -----------------------------------------------------------------------------------------*)
	(*Fault1501 - VFD01 Faulted*)
		Fault_Tmrs[1501].PT:= Short_Faults;
		Fault_Tmrs[1501]();
		Fault_Tmrs[1501].IN:= (GTAC_CONFIG.Option_VFD_Count>=1) AND
							MAIN.VFD01.Faulted;
		Out_To_ICxx.System_Faults[1501]:=Fault_Tmrs[1501].Q;
	(*Fault1502 - VFD02 Faulted*)
		Fault_Tmrs[1502].PT:= Short_Faults;
		Fault_Tmrs[1502]();
		Fault_Tmrs[1502].IN:= (GTAC_CONFIG.Option_VFD_Count>=2) AND
							MAIN.VFD02.Faulted;
		Out_To_ICxx.System_Faults[1502]:=Fault_Tmrs[1502].Q;
	(*Fault1503 - VFD03 Faulted*)
		Fault_Tmrs[1503].PT:= Short_Faults;
		Fault_Tmrs[1503]();
		Fault_Tmrs[1503].IN:= (GTAC_CONFIG.Option_VFD_Count>=3) AND
							MAIN.VFD03.Faulted;
		Out_To_ICxx.System_Faults[1503]:=Fault_Tmrs[1503].Q;
	(*Fault1504 - VFD04 Faulted*)
		Fault_Tmrs[1504].PT:= Short_Faults;
		Fault_Tmrs[1504]();
		Fault_Tmrs[1504].IN:= (GTAC_CONFIG.Option_VFD_Count>=4) AND
							MAIN.VFD04.Faulted;
		Out_To_ICxx.System_Faults[1504]:=Fault_Tmrs[1504].Q;
	(*Fault1505 - VFD05 Faulted*)
		Fault_Tmrs[1505].PT:= Short_Faults;
		Fault_Tmrs[1505]();
		Fault_Tmrs[1505].IN:= (GTAC_CONFIG.Option_VFD_Count>=5) AND
							MAIN.VFD05.Faulted;
		Out_To_ICxx.System_Faults[1505]:=Fault_Tmrs[1505].Q;
	
	

(*--------------------------------------------------------------------- Servo Drive General Fault Area ------------------------------------------------------*)

(*SDxx Axis 1 Faults*)

	(*Fault1531 - Servo Drive SD01 Axis1 Fault*)
		Fault_Tmrs[1531].PT:= Short_Faults;
		Fault_Tmrs[1531]();
		Fault_Tmrs[1531].IN:= Servo_Motion.SD[1].In_Error[1] OR Servo_Motion.SD[1].Discrete_Image.Safety_DIAG.bError;
		Out_To_ICxx.System_Faults[1531]:=Fault_Tmrs[1531].Q;
	(*Fault1532 - Servo Drive SD02 Axis1 Fault*)
		Fault_Tmrs[1532].PT:= Short_Faults;
		Fault_Tmrs[1532]();
		Fault_Tmrs[1532].IN:= Servo_Motion.SD[2].In_Error[1] OR Servo_Motion.SD[2].Discrete_Image.Safety_DIAG.bError;
		Out_To_ICxx.System_Faults[1532]:=Fault_Tmrs[1532].Q;
	(*Fault1533 - Servo Drive SD03 Axis1 Fault*)
		Fault_Tmrs[1533].PT:= Short_Faults;
		Fault_Tmrs[1533]();
		Fault_Tmrs[1533].IN:= Servo_Motion.SD[3].In_Error[1] OR Servo_Motion.SD[3].Discrete_Image.Safety_DIAG.bError;
		Out_To_ICxx.System_Faults[1533]:=Fault_Tmrs[1533].Q;
	(*Fault1534 - Servo Drive SD04 Axis1 Fault*)
		Fault_Tmrs[1534].PT:= Short_Faults;
		Fault_Tmrs[1534]();
		Fault_Tmrs[1534].IN:= Servo_Motion.SD[4].In_Error[1] OR Servo_Motion.SD[4].Discrete_Image.Safety_DIAG.bError;
		Out_To_ICxx.System_Faults[1534]:=Fault_Tmrs[1534].Q;
	(*Fault1535 - Servo Drive SD05 Axis1 Fault*)
		Fault_Tmrs[1535].PT:= Short_Faults;
		Fault_Tmrs[1535]();
		Fault_Tmrs[1535].IN:= Servo_Motion.SD[5].In_Error[1] OR Servo_Motion.SD[5].Discrete_Image.Safety_DIAG.bError;
		Out_To_ICxx.System_Faults[1535]:=Fault_Tmrs[1535].Q;
	(*Fault1536 - Servo Drive SD06 Axis1 Fault*)
		Fault_Tmrs[1536].PT:= Short_Faults;
		Fault_Tmrs[1536]();
		Fault_Tmrs[1536].IN:= Servo_Motion.SD[6].In_Error[1] OR Servo_Motion.SD[6].Discrete_Image.Safety_DIAG.bError;
		Out_To_ICxx.System_Faults[1536]:=Fault_Tmrs[1536].Q;
	(*Fault1537 - Servo Drive SD07 Axis1 Fault*)
		Fault_Tmrs[1537].PT:= Short_Faults;
		Fault_Tmrs[1537]();
		Fault_Tmrs[1537].IN:= Servo_Motion.SD[7].In_Error[1] OR Servo_Motion.SD[7].Discrete_Image.Safety_DIAG.bError;
		Out_To_ICxx.System_Faults[1537]:=Fault_Tmrs[1537].Q;
	(*Fault1538 - Servo Drive SD08 Axis1 Fault*)
		Fault_Tmrs[1538].PT:= Short_Faults;
		Fault_Tmrs[1538]();
		Fault_Tmrs[1538].IN:= Servo_Motion.SD[8].In_Error[1] OR Servo_Motion.SD[8].Discrete_Image.Safety_DIAG.bError;
		Out_To_ICxx.System_Faults[1538]:=Fault_Tmrs[1538].Q;
	(*Fault1539 - Servo Drive SD09 Axis1 Fault*)
		Fault_Tmrs[1539].PT:= Short_Faults;
		Fault_Tmrs[1539]();
		Fault_Tmrs[1539].IN:= Servo_Motion.SD[9].In_Error[1] OR Servo_Motion.SD[9].Discrete_Image.Safety_DIAG.bError;
		Out_To_ICxx.System_Faults[1539]:=Fault_Tmrs[1539].Q;
	(*Fault1540 - Servo Drive SD10 Axis1 Fault*)
		Fault_Tmrs[1540].PT:= Short_Faults;
		Fault_Tmrs[1540]();
		Fault_Tmrs[1540].IN:= Servo_Motion.SD[10].In_Error[1] OR Servo_Motion.SD[10].Discrete_Image.Safety_DIAG.bError;
		Out_To_ICxx.System_Faults[1540]:=Fault_Tmrs[1540].Q;
	(*Fault1541 - Servo Drive SD11 Axis1 Fault*)
		Fault_Tmrs[1541].PT:= Short_Faults;
		Fault_Tmrs[1541]();
		Fault_Tmrs[1541].IN:= Servo_Motion.SD[11].In_Error[1] OR Servo_Motion.SD[11].Discrete_Image.Safety_DIAG.bError;
		Out_To_ICxx.System_Faults[1541]:=Fault_Tmrs[1541].Q;
	(*Fault1542 - Servo Drive SD12 Axis1 Fault*)
		Fault_Tmrs[1542].PT:= Short_Faults;
		Fault_Tmrs[1542]();
		Fault_Tmrs[1542].IN:= Servo_Motion.SD[12].In_Error[1] OR Servo_Motion.SD[12].Discrete_Image.Safety_DIAG.bError;
		Out_To_ICxx.System_Faults[1542]:=Fault_Tmrs[1542].Q;
	(*Fault1543 - Servo Drive SD13 Axis1 Fault*)
		Fault_Tmrs[1543].PT:= Short_Faults;
		Fault_Tmrs[1543]();
		Fault_Tmrs[1543].IN:= Servo_Motion.SD[13].In_Error[1] OR Servo_Motion.SD[13].Discrete_Image.Safety_DIAG.bError;
		Out_To_ICxx.System_Faults[1543]:=Fault_Tmrs[1543].Q;
	(*Fault1544 - Servo Drive SD14 Axis1 Fault*)
		Fault_Tmrs[1544].PT:= Short_Faults;
		Fault_Tmrs[1544]();
		Fault_Tmrs[1544].IN:= Servo_Motion.SD[14].In_Error[1] OR Servo_Motion.SD[14].Discrete_Image.Safety_DIAG.bError;
		Out_To_ICxx.System_Faults[1544]:=Fault_Tmrs[1544].Q;
	(*Fault1545 - Servo Drive SD15 Axis1Fault*)
		Fault_Tmrs[1545].PT:= Short_Faults;
		Fault_Tmrs[1545]();
		Fault_Tmrs[1545].IN:= Servo_Motion.SD[15].In_Error[1] OR Servo_Motion.SD[15].Discrete_Image.Safety_DIAG.bError;
		Out_To_ICxx.System_Faults[1545]:=Fault_Tmrs[1545].Q;
	(*Fault1546 - Servo Drive SD16 Axis1 Fault*)
		Fault_Tmrs[1546].PT:= Short_Faults;
		Fault_Tmrs[1546]();
		Fault_Tmrs[1546].IN:= Servo_Motion.SD[16].In_Error[1] OR Servo_Motion.SD[16].Discrete_Image.Safety_DIAG.bError;
		Out_To_ICxx.System_Faults[1546]:=Fault_Tmrs[1546].Q;
	(*Fault1547 - Servo Drive SD17 Axis1 Fault*)
		Fault_Tmrs[1547].PT:= Short_Faults;
		Fault_Tmrs[1547]();
		Fault_Tmrs[1547].IN:= Servo_Motion.SD[17].In_Error[1] OR Servo_Motion.SD[17].Discrete_Image.Safety_DIAG.bError;
		Out_To_ICxx.System_Faults[1547]:=Fault_Tmrs[1547].Q;
	(*Fault1548 - Servo Drive SD18 Axis1 Fault*)
		Fault_Tmrs[1548].PT:= Short_Faults;
		Fault_Tmrs[1548]();
		Fault_Tmrs[1548].IN:= Servo_Motion.SD[18].In_Error[1] OR Servo_Motion.SD[18].Discrete_Image.Safety_DIAG.bError;
		Out_To_ICxx.System_Faults[1548]:=Fault_Tmrs[1548].Q;
	(*Fault1549 - Servo Drive SD19 Axis1 Fault*)
		Fault_Tmrs[1549].PT:= Short_Faults;
		Fault_Tmrs[1549]();
		Fault_Tmrs[1549].IN:= Servo_Motion.SD[19].In_Error[1] OR Servo_Motion.SD[19].Discrete_Image.Safety_DIAG.bError;
		Out_To_ICxx.System_Faults[1549]:=Fault_Tmrs[1549].Q;
	(*Fault1550 - Servo Drive SD20 Axis1 Fault*)
		Fault_Tmrs[1550].PT:= Short_Faults;
		Fault_Tmrs[1550]();
		Fault_Tmrs[1550].IN:= Servo_Motion.SD[20].In_Error[1] OR Servo_Motion.SD[20].Discrete_Image.Safety_DIAG.bError;
		Out_To_ICxx.System_Faults[1550]:=Fault_Tmrs[1550].Q;
	(*Fault1551 - Servo Drive SD21 Axis1 Fault*)
		Fault_Tmrs[1551].PT:= Short_Faults;
		Fault_Tmrs[1551]();
		Fault_Tmrs[1551].IN:= Servo_Motion.SD[21].In_Error[1] OR Servo_Motion.SD[21].Discrete_Image.Safety_DIAG.bError;
		Out_To_ICxx.System_Faults[1551]:=Fault_Tmrs[1551].Q;
	(*Fault1552 - Servo Drive SD22 Axis1 Fault*)
		Fault_Tmrs[1552].PT:= Short_Faults;
		Fault_Tmrs[1552]();
		Fault_Tmrs[1552].IN:= Servo_Motion.SD[22].In_Error[1] OR Servo_Motion.SD[22].Discrete_Image.Safety_DIAG.bError;
		Out_To_ICxx.System_Faults[1552]:=Fault_Tmrs[1552].Q;
	(*Fault1553 - Servo Drive SD23 Axis1 Fault*)
		Fault_Tmrs[1553].PT:= Short_Faults;
		Fault_Tmrs[1553]();
		Fault_Tmrs[1553].IN:= Servo_Motion.SD[23].In_Error[1] OR Servo_Motion.SD[23].Discrete_Image.Safety_DIAG.bError;
		Out_To_ICxx.System_Faults[1553]:=Fault_Tmrs[1553].Q;
	(*Fault1554 - Servo Drive SD24 Axis1 Fault*)
		Fault_Tmrs[1554].PT:= Short_Faults;
		Fault_Tmrs[1554]();
		Fault_Tmrs[1554].IN:= Servo_Motion.SD[24].In_Error[1] OR Servo_Motion.SD[24].Discrete_Image.Safety_DIAG.bError;
		Out_To_ICxx.System_Faults[1554]:=Fault_Tmrs[1554].Q;
	(*Fault1555 - Servo Drive SD25 Axis1 Fault*)
		Fault_Tmrs[1555].PT:= Short_Faults;
		Fault_Tmrs[1555]();
		Fault_Tmrs[1555].IN:= Servo_Motion.SD[25].In_Error[1] OR Servo_Motion.SD[25].Discrete_Image.Safety_DIAG.bError;
		Out_To_ICxx.System_Faults[1555]:=Fault_Tmrs[1555].Q;
	(*Fault1556 - Servo Drive SD26 Axis1 Fault*)
		Fault_Tmrs[1556].PT:= Short_Faults;
		Fault_Tmrs[1556]();
		Fault_Tmrs[1556].IN:= Servo_Motion.SD[26].In_Error[1] OR Servo_Motion.SD[26].Discrete_Image.Safety_DIAG.bError;
		Out_To_ICxx.System_Faults[1556]:=Fault_Tmrs[1556].Q;
	(*Fault1557 - Servo Drive SD27 Axis1 Fault*)
		Fault_Tmrs[1557].PT:= Short_Faults;
		Fault_Tmrs[1557]();
		Fault_Tmrs[1557].IN:= Servo_Motion.SD[27].In_Error[1] OR Servo_Motion.SD[27].Discrete_Image.Safety_DIAG.bError;
		Out_To_ICxx.System_Faults[1557]:=Fault_Tmrs[1557].Q;
	(*Fault1558 - Servo Drive SD28 Axis1 Fault*)
		Fault_Tmrs[1558].PT:= Short_Faults;
		Fault_Tmrs[1558]();
		Fault_Tmrs[1558].IN:= Servo_Motion.SD[28].In_Error[1] OR Servo_Motion.SD[28].Discrete_Image.Safety_DIAG.bError;
		Out_To_ICxx.System_Faults[1558]:=Fault_Tmrs[1558].Q;
	(*Fault1559 - Servo Drive SD29 Axis1 Fault*)
		Fault_Tmrs[1559].PT:= Short_Faults;
		Fault_Tmrs[1559]();
		Fault_Tmrs[1559].IN:= Servo_Motion.SD[29].In_Error[1] OR Servo_Motion.SD[29].Discrete_Image.Safety_DIAG.bError;
		Out_To_ICxx.System_Faults[1559]:=Fault_Tmrs[1559].Q;
	(*Fault1560 - Servo Drive SD30 Axis1 Fault*)
		Fault_Tmrs[1560].PT:= Short_Faults;
		Fault_Tmrs[1560]();
		Fault_Tmrs[1560].IN:= Servo_Motion.SD[30].In_Error[1] OR Servo_Motion.SD[30].Discrete_Image.Safety_DIAG.bError;
		Out_To_ICxx.System_Faults[1560]:=Fault_Tmrs[1560].Q;

(*SDxx Axis 2 Faults*)

	(*Fault1561 - Servo Drive SD01 Axis2 Fault*)
		Fault_Tmrs[1561].PT:= Short_Faults;
		Fault_Tmrs[1561]();
		Fault_Tmrs[1561].IN:= Servo_Motion.SD[1].In_Error[2] OR Servo_Motion.SD[1].Discrete_Image.Safety_DIAG.bError;
		Out_To_ICxx.System_Faults[1561]:=Fault_Tmrs[1561].Q;
	(*Fault1562 - Servo Drive SD02 Axis2 Fault*)
		Fault_Tmrs[1562].PT:= Short_Faults;
		Fault_Tmrs[1562]();
		Fault_Tmrs[1562].IN:= Servo_Motion.SD[2].In_Error[2] OR Servo_Motion.SD[2].Discrete_Image.Safety_DIAG.bError;
		Out_To_ICxx.System_Faults[1562]:=Fault_Tmrs[1562].Q;
	(*Fault1563 - Servo Drive SD03 Axis2 Fault*)
		Fault_Tmrs[1563].PT:= Short_Faults;
		Fault_Tmrs[1563]();
		Fault_Tmrs[1563].IN:= Servo_Motion.SD[3].In_Error[2] OR Servo_Motion.SD[3].Discrete_Image.Safety_DIAG.bError;
		Out_To_ICxx.System_Faults[1563]:=Fault_Tmrs[1563].Q;
	(*Fault1564 - Servo Drive SD04 Axis2 Fault*)
		Fault_Tmrs[1564].PT:= Short_Faults;
		Fault_Tmrs[1564]();
		Fault_Tmrs[1564].IN:= Servo_Motion.SD[4].In_Error[2] OR Servo_Motion.SD[4].Discrete_Image.Safety_DIAG.bError;
		Out_To_ICxx.System_Faults[1564]:=Fault_Tmrs[1564].Q;
	(*Fault1565 - Servo Drive SD05 Axis2 Fault*)
		Fault_Tmrs[1565].PT:= Short_Faults;
		Fault_Tmrs[1565]();
		Fault_Tmrs[1565].IN:= Servo_Motion.SD[5].In_Error[2] OR Servo_Motion.SD[5].Discrete_Image.Safety_DIAG.bError;
		Out_To_ICxx.System_Faults[1565]:=Fault_Tmrs[1565].Q;
	(*Fault1566 - Servo Drive SD06 Axis2 Fault*)
		Fault_Tmrs[1566].PT:= Short_Faults;
		Fault_Tmrs[1566]();
		Fault_Tmrs[1566].IN:= Servo_Motion.SD[6].In_Error[2] OR Servo_Motion.SD[6].Discrete_Image.Safety_DIAG.bError;
		Out_To_ICxx.System_Faults[1566]:=Fault_Tmrs[1566].Q;
	(*Fault1567 - Servo Drive SD07 Axis2 Fault*)
		Fault_Tmrs[1567].PT:= Short_Faults;
		Fault_Tmrs[1567]();
		Fault_Tmrs[1567].IN:= Servo_Motion.SD[7].In_Error[2] OR Servo_Motion.SD[7].Discrete_Image.Safety_DIAG.bError;
		Out_To_ICxx.System_Faults[1567]:=Fault_Tmrs[1567].Q;
	(*Fault1568 - Servo Drive SD08 Axis2 Fault*)
		Fault_Tmrs[1568].PT:= Short_Faults;
		Fault_Tmrs[1568]();
		Fault_Tmrs[1568].IN:= Servo_Motion.SD[8].In_Error[2] OR Servo_Motion.SD[8].Discrete_Image.Safety_DIAG.bError;
		Out_To_ICxx.System_Faults[1568]:=Fault_Tmrs[1568].Q;
	(*Fault1569 - Servo Drive SD09 Axis2 Fault*)
		Fault_Tmrs[1569].PT:= Short_Faults;
		Fault_Tmrs[1569]();
		Fault_Tmrs[1569].IN:= Servo_Motion.SD[9].In_Error[2] OR Servo_Motion.SD[9].Discrete_Image.Safety_DIAG.bError;
		Out_To_ICxx.System_Faults[1569]:=Fault_Tmrs[1569].Q;
	(*Fault1570 - Servo Drive SD10 Axis2 Fault*)
		Fault_Tmrs[1570].PT:= Short_Faults;
		Fault_Tmrs[1570]();
		Fault_Tmrs[1570].IN:= Servo_Motion.SD[10].In_Error[2] OR Servo_Motion.SD[10].Discrete_Image.Safety_DIAG.bError;
		Out_To_ICxx.System_Faults[1570]:=Fault_Tmrs[1570].Q;
	(*Fault1571 - Servo Drive SD11 Axis2 Fault*)
		Fault_Tmrs[1571].PT:= Short_Faults;
		Fault_Tmrs[1571]();
		Fault_Tmrs[1571].IN:= Servo_Motion.SD[11].In_Error[2] OR Servo_Motion.SD[11].Discrete_Image.Safety_DIAG.bError;
		Out_To_ICxx.System_Faults[1571]:=Fault_Tmrs[1571].Q;
	(*Fault1572 - Servo Drive SD12 Axis2 Fault*)
		Fault_Tmrs[1572].PT:= Short_Faults;
		Fault_Tmrs[1572]();
		Fault_Tmrs[1572].IN:= Servo_Motion.SD[12].In_Error[2] OR Servo_Motion.SD[12].Discrete_Image.Safety_DIAG.bError;
		Out_To_ICxx.System_Faults[1572]:=Fault_Tmrs[1572].Q;
	(*Fault1573 - Servo Drive SD13 Axis2 Fault*)
		Fault_Tmrs[1573].PT:= Short_Faults;
		Fault_Tmrs[1573]();
		Fault_Tmrs[1573].IN:= Servo_Motion.SD[13].In_Error[2] OR Servo_Motion.SD[13].Discrete_Image.Safety_DIAG.bError;
		Out_To_ICxx.System_Faults[1573]:=Fault_Tmrs[1573].Q;
	(*Fault1574 - Servo Drive SD14 Axis2 Fault*)
		Fault_Tmrs[1574].PT:= Short_Faults;
		Fault_Tmrs[1574]();
		Fault_Tmrs[1574].IN:= Servo_Motion.SD[14].In_Error[2] OR Servo_Motion.SD[14].Discrete_Image.Safety_DIAG.bError;
		Out_To_ICxx.System_Faults[1574]:=Fault_Tmrs[1574].Q;
	(*Fault1575 - Servo Drive SD15 Axis2 Fault*)
		Fault_Tmrs[1575].PT:= Short_Faults;
		Fault_Tmrs[1575]();
		Fault_Tmrs[1575].IN:= Servo_Motion.SD[15].In_Error[2] OR Servo_Motion.SD[15].Discrete_Image.Safety_DIAG.bError;
		Out_To_ICxx.System_Faults[1575]:=Fault_Tmrs[1575].Q;
	(*Fault1576 - Servo Drive SD16 Axis2 Fault*)
		Fault_Tmrs[1576].PT:= Short_Faults;
		Fault_Tmrs[1576]();
		Fault_Tmrs[1576].IN:= Servo_Motion.SD[16].In_Error[2] OR Servo_Motion.SD[16].Discrete_Image.Safety_DIAG.bError;
		Out_To_ICxx.System_Faults[1576]:=Fault_Tmrs[1576].Q;
	(*Fault1577 - Servo Drive SD17 Axis2 Fault*)
		Fault_Tmrs[1577].PT:= Short_Faults;
		Fault_Tmrs[1577]();
		Fault_Tmrs[1577].IN:= Servo_Motion.SD[17].In_Error[2] OR Servo_Motion.SD[17].Discrete_Image.Safety_DIAG.bError;
		Out_To_ICxx.System_Faults[1577]:=Fault_Tmrs[1577].Q;
	(*Fault1578 - Servo Drive SD18 Axis2 Fault*)
		Fault_Tmrs[1578].PT:= Short_Faults;
		Fault_Tmrs[1578]();
		Fault_Tmrs[1578].IN:= Servo_Motion.SD[18].In_Error[2] OR Servo_Motion.SD[18].Discrete_Image.Safety_DIAG.bError;
		Out_To_ICxx.System_Faults[1578]:=Fault_Tmrs[1578].Q;
	(*Fault1579 - Servo Drive SD19 Axis2 Fault*)
		Fault_Tmrs[1579].PT:= Short_Faults;
		Fault_Tmrs[1579]();
		Fault_Tmrs[1579].IN:= Servo_Motion.SD[19].In_Error[2] OR Servo_Motion.SD[19].Discrete_Image.Safety_DIAG.bError;
		Out_To_ICxx.System_Faults[1579]:=Fault_Tmrs[1579].Q;
	(*Fault1580 - Servo Drive SD20 Axis2 Fault*)
		Fault_Tmrs[1580].PT:= Short_Faults;
		Fault_Tmrs[1580]();
		Fault_Tmrs[1580].IN:= Servo_Motion.SD[20].In_Error[2] OR Servo_Motion.SD[20].Discrete_Image.Safety_DIAG.bError;
		Out_To_ICxx.System_Faults[1580]:=Fault_Tmrs[1580].Q;
	(*Fault1581 - Servo Drive SD21 Axis2 Fault*)
		Fault_Tmrs[1581].PT:= Short_Faults;
		Fault_Tmrs[1581]();
		Fault_Tmrs[1581].IN:= Servo_Motion.SD[21].In_Error[2] OR Servo_Motion.SD[21].Discrete_Image.Safety_DIAG.bError;
		Out_To_ICxx.System_Faults[1581]:=Fault_Tmrs[1581].Q;
	(*Fault1582 - Servo Drive SD22 Axis2 Fault*)
		Fault_Tmrs[1582].PT:= Short_Faults;
		Fault_Tmrs[1582]();
		Fault_Tmrs[1582].IN:= Servo_Motion.SD[22].In_Error[2] OR Servo_Motion.SD[22].Discrete_Image.Safety_DIAG.bError;
		Out_To_ICxx.System_Faults[1582]:=Fault_Tmrs[1582].Q;
	(*Fault1583 - Servo Drive SD23 Axis2 Fault*)
		Fault_Tmrs[1583].PT:= Short_Faults;
		Fault_Tmrs[1583]();
		Fault_Tmrs[1583].IN:= Servo_Motion.SD[23].In_Error[2] OR Servo_Motion.SD[23].Discrete_Image.Safety_DIAG.bError;
		Out_To_ICxx.System_Faults[1583]:=Fault_Tmrs[1583].Q;
	(*Fault1584 - Servo Drive SD24 Axis2 Fault*)
		Fault_Tmrs[1584].PT:= Short_Faults;
		Fault_Tmrs[1584]();
		Fault_Tmrs[1584].IN:= Servo_Motion.SD[24].In_Error[2] OR Servo_Motion.SD[24].Discrete_Image.Safety_DIAG.bError;
		Out_To_ICxx.System_Faults[1584]:=Fault_Tmrs[1584].Q;
	(*Fault1585 - Servo Drive SD25 Axis2 Fault*)
		Fault_Tmrs[1585].PT:= Short_Faults;
		Fault_Tmrs[1585]();
		Fault_Tmrs[1585].IN:= Servo_Motion.SD[25].In_Error[2] OR Servo_Motion.SD[25].Discrete_Image.Safety_DIAG.bError;
		Out_To_ICxx.System_Faults[1585]:=Fault_Tmrs[1585].Q;
	(*Fault1586 - Servo Drive SD26 Axis2 Fault*)
		Fault_Tmrs[1586].PT:= Short_Faults;
		Fault_Tmrs[1586]();
		Fault_Tmrs[1586].IN:= Servo_Motion.SD[26].In_Error[2] OR Servo_Motion.SD[26].Discrete_Image.Safety_DIAG.bError;
		Out_To_ICxx.System_Faults[1586]:=Fault_Tmrs[1586].Q;
	(*Fault1587 - Servo Drive SD27 Axis2 Fault*)
		Fault_Tmrs[1587].PT:= Short_Faults;
		Fault_Tmrs[1587]();
		Fault_Tmrs[1587].IN:= Servo_Motion.SD[27].In_Error[2] OR Servo_Motion.SD[27].Discrete_Image.Safety_DIAG.bError;
		Out_To_ICxx.System_Faults[1587]:=Fault_Tmrs[1587].Q;
	(*Fault1588 - Servo Drive SD28 Axis2 Fault*)
		Fault_Tmrs[1588].PT:= Short_Faults;
		Fault_Tmrs[1588]();
		Fault_Tmrs[1588].IN:= Servo_Motion.SD[28].In_Error[2] OR Servo_Motion.SD[28].Discrete_Image.Safety_DIAG.bError;
		Out_To_ICxx.System_Faults[1588]:=Fault_Tmrs[1588].Q;
	(*Fault1589 - Servo Drive SD29 Axis2 Fault*)
		Fault_Tmrs[1589].PT:= Short_Faults;
		Fault_Tmrs[1589]();
		Fault_Tmrs[1589].IN:= Servo_Motion.SD[29].In_Error[2] OR Servo_Motion.SD[29].Discrete_Image.Safety_DIAG.bError;
		Out_To_ICxx.System_Faults[1589]:=Fault_Tmrs[1589].Q;
	(*Fault1590 - Servo Drive SD30 Axis2 Fault*)
		Fault_Tmrs[1590].PT:= Short_Faults;
		Fault_Tmrs[1590]();
		Fault_Tmrs[1590].IN:= Servo_Motion.SD[30].In_Error[2] OR Servo_Motion.SD[30].Discrete_Image.Safety_DIAG.bError;
		Out_To_ICxx.System_Faults[1590]:=Fault_Tmrs[1590].Q;


	(*--------------------------------------------------------------------- General Minor Fault Area ------------------------------------------------------*)

	(*Fault1561 - spare misc fault*)
		Fault_Tmrs[1591].PT:= Short_Faults;
		Fault_Tmrs[1591]();
		Fault_Tmrs[1591].IN:= FALSE;
		Out_To_ICxx.System_Faults[1591]:=Fault_Tmrs[1591].Q;
	(*.............................*)
	(*.............................*)
	(*.............................*)
	(*Fault1639 - spare misc fault*)
		Fault_Tmrs[1639].PT:= Short_Faults;
		Fault_Tmrs[1639]();
		Fault_Tmrs[1639].IN:= FALSE;
		Out_To_ICxx.System_Faults[1639]:=Fault_Tmrs[1639].Q;


END_IF; (*End of Configuration Condition Check*)


(*-----------------------------------------------------------------------------------------------------------------------------------------------------------------------------------------------*)
(*----------------------------- Generate General Control System Fault to Drive Red Flashing Prompt on UI -------------------------------------------------*)

(*Drive Flags Generate UI Prompting on Controls Menu Screen*)
	(*System Related Faults*)
	Out_To_ICxx.ICxx_UI_FaultPrompts.0:=
		Out_To_ICxx.System_Faults[2]		(*Main Board CPU Over Temp*)
		OR Out_To_ICxx.System_Faults[3];	(*ECAT Master bad DevState*)
	(*IC01*)
	Out_To_ICxx.ICxx_UI_FaultPrompts.1:=
		Out_To_ICxx.ICxx_UI_FaultPrompts.0	(*Include IC01 IPC system faults*)
		OR Out_To_ICxx.System_Faults[141]
		OR Out_To_ICxx.System_Faults[142]
		OR Out_To_ICxx.System_Faults[143]
		OR Out_To_ICxx.System_Faults[144]
		OR Out_To_ICxx.System_Faults[591]
		OR Out_To_ICxx.System_Faults[601]
		OR Out_To_ICxx.System_Faults[602]
		OR Out_To_ICxx.ICxx_UI_FaultPrompts.0;	(*Include SMB /ECAT Master Faults on IC01 Prompting*)
	(*IC02*)
	Out_To_ICxx.ICxx_UI_FaultPrompts.2:=
		Out_To_ICxx.System_Faults[151]
		OR Out_To_ICxx.System_Faults[152]
		OR Out_To_ICxx.System_Faults[153]
		OR Out_To_ICxx.System_Faults[154]
		OR Out_To_ICxx.System_Faults[592]
		OR Out_To_ICxx.System_Faults[603]
		OR Out_To_ICxx.System_Faults[604];
	(*IC03*)
	Out_To_ICxx.ICxx_UI_FaultPrompts.3:=
		Out_To_ICxx.System_Faults[161]
		OR Out_To_ICxx.System_Faults[162]
		OR Out_To_ICxx.System_Faults[163]
		OR Out_To_ICxx.System_Faults[164]
		OR Out_To_ICxx.System_Faults[593]
		OR Out_To_ICxx.System_Faults[605]
		OR Out_To_ICxx.System_Faults[606];
	(*IC04*)
	Out_To_ICxx.ICxx_UI_FaultPrompts.4:=
		Out_To_ICxx.System_Faults[171]
		OR Out_To_ICxx.System_Faults[172]
		OR Out_To_ICxx.System_Faults[173]
		OR Out_To_ICxx.System_Faults[174]
		OR Out_To_ICxx.System_Faults[594]
		OR Out_To_ICxx.System_Faults[607]
		OR Out_To_ICxx.System_Faults[608];
	(*IC05*)
	Out_To_ICxx.ICxx_UI_FaultPrompts.5:=
		Out_To_ICxx.System_Faults[181]
		OR Out_To_ICxx.System_Faults[182]
		OR Out_To_ICxx.System_Faults[183]
		OR Out_To_ICxx.System_Faults[184]
		OR Out_To_ICxx.System_Faults[595]
		OR Out_To_ICxx.System_Faults[609]
		OR Out_To_ICxx.System_Faults[610];
	(*IC06*)
	Out_To_ICxx.ICxx_UI_FaultPrompts.6:=
		Out_To_ICxx.System_Faults[191]
		OR Out_To_ICxx.System_Faults[192]
		OR Out_To_ICxx.System_Faults[193]
		OR Out_To_ICxx.System_Faults[194]
		OR Out_To_ICxx.System_Faults[596]
		OR Out_To_ICxx.System_Faults[611]
		OR Out_To_ICxx.System_Faults[612];
	(*IC07*)
	Out_To_ICxx.ICxx_UI_FaultPrompts.7:=
		Out_To_ICxx.System_Faults[201]
		OR Out_To_ICxx.System_Faults[202]
		OR Out_To_ICxx.System_Faults[203]
		OR Out_To_ICxx.System_Faults[204]
		OR Out_To_ICxx.System_Faults[597]
		OR Out_To_ICxx.System_Faults[613]
		OR Out_To_ICxx.System_Faults[614];
	(*IC08*)
	Out_To_ICxx.ICxx_UI_FaultPrompts.8:=
		Out_To_ICxx.System_Faults[211]
		OR Out_To_ICxx.System_Faults[212]
		OR Out_To_ICxx.System_Faults[213]
		OR Out_To_ICxx.System_Faults[214]
		OR Out_To_ICxx.System_Faults[598]
		OR Out_To_ICxx.System_Faults[615]
		OR Out_To_ICxx.System_Faults[616];

	(*IC01-TSAFE ONLY*)
	Out_To_ICxx.ICxx_UI_FaultPrompts.11:=
		Out_To_ICxx.System_Faults[141]
		OR Out_To_ICxx.System_Faults[142]
		OR Out_To_ICxx.System_Faults[143]
		OR Out_To_ICxx.System_Faults[144];
	(*IC02-TSAFE ONLY*)
	Out_To_ICxx.ICxx_UI_FaultPrompts.12:=
		Out_To_ICxx.System_Faults[151]
		OR Out_To_ICxx.System_Faults[152]
		OR Out_To_ICxx.System_Faults[153]
		OR Out_To_ICxx.System_Faults[154];
	(*IC03-TSAFE ONLY*)
	Out_To_ICxx.ICxx_UI_FaultPrompts.13:=
		Out_To_ICxx.System_Faults[161]
		OR Out_To_ICxx.System_Faults[162]
		OR Out_To_ICxx.System_Faults[163]
		OR Out_To_ICxx.System_Faults[164];
	(*IC04-TSAFE ONLY*)
	Out_To_ICxx.ICxx_UI_FaultPrompts.14:=
		Out_To_ICxx.System_Faults[171]
		OR Out_To_ICxx.System_Faults[172]
		OR Out_To_ICxx.System_Faults[173]
		OR Out_To_ICxx.System_Faults[174];
	(*IC05-TSAFE ONLY*)
	Out_To_ICxx.ICxx_UI_FaultPrompts.15:=
		Out_To_ICxx.System_Faults[181]
		OR Out_To_ICxx.System_Faults[182]
		OR Out_To_ICxx.System_Faults[183]
		OR Out_To_ICxx.System_Faults[184];
	(*IC06-TSAFE ONLY*)
	Out_To_ICxx.ICxx_UI_FaultPrompts.16:=
		Out_To_ICxx.System_Faults[191]
		OR Out_To_ICxx.System_Faults[192]
		OR Out_To_ICxx.System_Faults[193]
		OR Out_To_ICxx.System_Faults[194];
	(*IC07-TSAFE ONLY*)
	Out_To_ICxx.ICxx_UI_FaultPrompts.17:=
		Out_To_ICxx.System_Faults[201]
		OR Out_To_ICxx.System_Faults[202]
		OR Out_To_ICxx.System_Faults[203]
		OR Out_To_ICxx.System_Faults[204];
	(*IC08-TSAFE ONLY*)
	Out_To_ICxx.ICxx_UI_FaultPrompts.18:=
		Out_To_ICxx.System_Faults[211]
		OR Out_To_ICxx.System_Faults[212]
		OR Out_To_ICxx.System_Faults[213]
		OR Out_To_ICxx.System_Faults[214];
	
		
		
	(*R1*)
	Out_To_ICxx.Rxx_UI_FaultPrompts.1:=
		Out_To_ICxx.System_Faults[221]
		OR Out_To_ICxx.System_Faults[222]
		OR Out_To_ICxx.System_Faults[223]
		OR Out_To_ICxx.System_Faults[224]
		OR Out_To_ICxx.System_Faults[631]
		OR Out_To_ICxx.System_Faults[661]
		OR Out_To_ICxx.System_Faults[691];
	(*R2*)
	Out_To_ICxx.Rxx_UI_FaultPrompts.2:=
		Out_To_ICxx.System_Faults[231]
		OR Out_To_ICxx.System_Faults[232]
		OR Out_To_ICxx.System_Faults[233]
		OR Out_To_ICxx.System_Faults[234]
		OR Out_To_ICxx.System_Faults[632]
		OR Out_To_ICxx.System_Faults[662]
		OR Out_To_ICxx.System_Faults[692];
	(*R3*)
	Out_To_ICxx.Rxx_UI_FaultPrompts.3:=
		Out_To_ICxx.System_Faults[241]
		OR Out_To_ICxx.System_Faults[242]
		OR Out_To_ICxx.System_Faults[243]
		OR Out_To_ICxx.System_Faults[244]
		OR Out_To_ICxx.System_Faults[633]
		OR Out_To_ICxx.System_Faults[663]
		OR Out_To_ICxx.System_Faults[693];
	(*R4*)
	Out_To_ICxx.Rxx_UI_FaultPrompts.4:=
		Out_To_ICxx.System_Faults[251]
		OR Out_To_ICxx.System_Faults[252]
		OR Out_To_ICxx.System_Faults[253]
		OR Out_To_ICxx.System_Faults[254]
		OR Out_To_ICxx.System_Faults[634]
		OR Out_To_ICxx.System_Faults[664]
		OR Out_To_ICxx.System_Faults[694];
	(*R5*)
	Out_To_ICxx.Rxx_UI_FaultPrompts.5:=
		Out_To_ICxx.System_Faults[261]
		OR Out_To_ICxx.System_Faults[262]
		OR Out_To_ICxx.System_Faults[263]
		OR Out_To_ICxx.System_Faults[264]
		OR Out_To_ICxx.System_Faults[635]
		OR Out_To_ICxx.System_Faults[665]
		OR Out_To_ICxx.System_Faults[695];
	(*R6*)
	Out_To_ICxx.Rxx_UI_FaultPrompts.6:=
		Out_To_ICxx.System_Faults[271]
		OR Out_To_ICxx.System_Faults[272]
		OR Out_To_ICxx.System_Faults[273]
		OR Out_To_ICxx.System_Faults[274]
		OR Out_To_ICxx.System_Faults[636]
		OR Out_To_ICxx.System_Faults[666]
		OR Out_To_ICxx.System_Faults[696];
	(*R7*)
	Out_To_ICxx.Rxx_UI_FaultPrompts.7:=
		Out_To_ICxx.System_Faults[281]
		OR Out_To_ICxx.System_Faults[282]
		OR Out_To_ICxx.System_Faults[283]
		OR Out_To_ICxx.System_Faults[284]
		OR Out_To_ICxx.System_Faults[637]
		OR Out_To_ICxx.System_Faults[667]
		OR Out_To_ICxx.System_Faults[697];
	(*R8*)
	Out_To_ICxx.Rxx_UI_FaultPrompts.8:=
		Out_To_ICxx.System_Faults[291]
		OR Out_To_ICxx.System_Faults[292]
		OR Out_To_ICxx.System_Faults[293]
		OR Out_To_ICxx.System_Faults[294]
		OR Out_To_ICxx.System_Faults[638]
		OR Out_To_ICxx.System_Faults[668]
		OR Out_To_ICxx.System_Faults[698];
	(*R9*)
	Out_To_ICxx.Rxx_UI_FaultPrompts.9:=
		Out_To_ICxx.System_Faults[301]
		OR Out_To_ICxx.System_Faults[302]
		OR Out_To_ICxx.System_Faults[303]
		OR Out_To_ICxx.System_Faults[304]
		OR Out_To_ICxx.System_Faults[639]
		OR Out_To_ICxx.System_Faults[669]
		OR Out_To_ICxx.System_Faults[699];
	(*R10*)
	Out_To_ICxx.Rxx_UI_FaultPrompts.10:=
		Out_To_ICxx.System_Faults[311]
		OR Out_To_ICxx.System_Faults[312]
		OR Out_To_ICxx.System_Faults[313]
		OR Out_To_ICxx.System_Faults[314]
		OR Out_To_ICxx.System_Faults[640]
		OR Out_To_ICxx.System_Faults[670]
		OR Out_To_ICxx.System_Faults[700];
	(*R11*)
	Out_To_ICxx.Rxx_UI_FaultPrompts.11:=
		Out_To_ICxx.System_Faults[321]
		OR Out_To_ICxx.System_Faults[322]
		OR Out_To_ICxx.System_Faults[323]
		OR Out_To_ICxx.System_Faults[324]
		OR Out_To_ICxx.System_Faults[641]
		OR Out_To_ICxx.System_Faults[671]
		OR Out_To_ICxx.System_Faults[701];
	(*R12*)
	Out_To_ICxx.Rxx_UI_FaultPrompts.12:=
		Out_To_ICxx.System_Faults[331]
		OR Out_To_ICxx.System_Faults[332]
		OR Out_To_ICxx.System_Faults[333]
		OR Out_To_ICxx.System_Faults[334]
		OR Out_To_ICxx.System_Faults[642]
		OR Out_To_ICxx.System_Faults[672]
		OR Out_To_ICxx.System_Faults[702];
	(*R13*)
	Out_To_ICxx.Rxx_UI_FaultPrompts.13:=
		Out_To_ICxx.System_Faults[341]
		OR Out_To_ICxx.System_Faults[342]
		OR Out_To_ICxx.System_Faults[343]
		OR Out_To_ICxx.System_Faults[344]
		OR Out_To_ICxx.System_Faults[643]
		OR Out_To_ICxx.System_Faults[673]
		OR Out_To_ICxx.System_Faults[703];
	(*R14*)
	Out_To_ICxx.Rxx_UI_FaultPrompts.14:=
		Out_To_ICxx.System_Faults[351]
		OR Out_To_ICxx.System_Faults[352]
		OR Out_To_ICxx.System_Faults[353]
		OR Out_To_ICxx.System_Faults[354]
		OR Out_To_ICxx.System_Faults[644]
		OR Out_To_ICxx.System_Faults[674]
		OR Out_To_ICxx.System_Faults[704];
	(*R15*)
	Out_To_ICxx.Rxx_UI_FaultPrompts.15:=
		Out_To_ICxx.System_Faults[361]
		OR Out_To_ICxx.System_Faults[362]
		OR Out_To_ICxx.System_Faults[363]
		OR Out_To_ICxx.System_Faults[364]
		OR Out_To_ICxx.System_Faults[655]
		OR Out_To_ICxx.System_Faults[675]
		OR Out_To_ICxx.System_Faults[705];
	(*R16*)
	Out_To_ICxx.Rxx_UI_FaultPrompts.16:=
		Out_To_ICxx.System_Faults[371]
		OR Out_To_ICxx.System_Faults[372]
		OR Out_To_ICxx.System_Faults[373]
		OR Out_To_ICxx.System_Faults[374]
		OR Out_To_ICxx.System_Faults[646]
		OR Out_To_ICxx.System_Faults[676]
		OR Out_To_ICxx.System_Faults[706];
	(*R17*)
	Out_To_ICxx.Rxx_UI_FaultPrompts.17:=
		Out_To_ICxx.System_Faults[381]
		OR Out_To_ICxx.System_Faults[382]
		OR Out_To_ICxx.System_Faults[383]
		OR Out_To_ICxx.System_Faults[384]
		OR Out_To_ICxx.System_Faults[647]
		OR Out_To_ICxx.System_Faults[677]
		OR Out_To_ICxx.System_Faults[707];
	(*R18*)
	Out_To_ICxx.Rxx_UI_FaultPrompts.18:=
		Out_To_ICxx.System_Faults[391]
		OR Out_To_ICxx.System_Faults[392]
		OR Out_To_ICxx.System_Faults[393]
		OR Out_To_ICxx.System_Faults[394]
		OR Out_To_ICxx.System_Faults[648]
		OR Out_To_ICxx.System_Faults[678]
		OR Out_To_ICxx.System_Faults[708];
	(*R19*)
	Out_To_ICxx.Rxx_UI_FaultPrompts.19:=
		Out_To_ICxx.System_Faults[401]
		OR Out_To_ICxx.System_Faults[402]
		OR Out_To_ICxx.System_Faults[403]
		OR Out_To_ICxx.System_Faults[404]
		OR Out_To_ICxx.System_Faults[649]
		OR Out_To_ICxx.System_Faults[679]
		OR Out_To_ICxx.System_Faults[709];
	(*R20*)
	Out_To_ICxx.Rxx_UI_FaultPrompts.20:=
		Out_To_ICxx.System_Faults[411]
		OR Out_To_ICxx.System_Faults[412]
		OR Out_To_ICxx.System_Faults[413]
		OR Out_To_ICxx.System_Faults[414]
		OR Out_To_ICxx.System_Faults[650]
		OR Out_To_ICxx.System_Faults[680]
		OR Out_To_ICxx.System_Faults[710];
	(*R21*)
	Out_To_ICxx.Rxx_UI_FaultPrompts.21:=
		Out_To_ICxx.System_Faults[421]
		OR Out_To_ICxx.System_Faults[422]
		OR Out_To_ICxx.System_Faults[423]
		OR Out_To_ICxx.System_Faults[424]
		OR Out_To_ICxx.System_Faults[651]
		OR Out_To_ICxx.System_Faults[681]
		OR Out_To_ICxx.System_Faults[711];
	(*R22*)
	Out_To_ICxx.Rxx_UI_FaultPrompts.22:=
		Out_To_ICxx.System_Faults[431]
		OR Out_To_ICxx.System_Faults[432]
		OR Out_To_ICxx.System_Faults[433]
		OR Out_To_ICxx.System_Faults[434]
		OR Out_To_ICxx.System_Faults[652]
		OR Out_To_ICxx.System_Faults[682]
		OR Out_To_ICxx.System_Faults[712];
	(*R23*)
	Out_To_ICxx.Rxx_UI_FaultPrompts.23:=
		Out_To_ICxx.System_Faults[441]
		OR Out_To_ICxx.System_Faults[442]
		OR Out_To_ICxx.System_Faults[443]
		OR Out_To_ICxx.System_Faults[444]
		OR Out_To_ICxx.System_Faults[653]
		OR Out_To_ICxx.System_Faults[683]
		OR Out_To_ICxx.System_Faults[713];
	(*R24*)
	Out_To_ICxx.Rxx_UI_FaultPrompts.24:=
		Out_To_ICxx.System_Faults[451]
		OR Out_To_ICxx.System_Faults[452]
		OR Out_To_ICxx.System_Faults[453]
		OR Out_To_ICxx.System_Faults[454]
		OR Out_To_ICxx.System_Faults[654]
		OR Out_To_ICxx.System_Faults[684]
		OR Out_To_ICxx.System_Faults[714];
	(*R25*)
	Out_To_ICxx.Rxx_UI_FaultPrompts.25:=
		Out_To_ICxx.System_Faults[461]
		OR Out_To_ICxx.System_Faults[462]
		OR Out_To_ICxx.System_Faults[463]
		OR Out_To_ICxx.System_Faults[464]
		OR Out_To_ICxx.System_Faults[655]
		OR Out_To_ICxx.System_Faults[685]
		OR Out_To_ICxx.System_Faults[715];
	(*R26*)
	Out_To_ICxx.Rxx_UI_FaultPrompts.26:=
		Out_To_ICxx.System_Faults[471]
		OR Out_To_ICxx.System_Faults[472]
		OR Out_To_ICxx.System_Faults[473]
		OR Out_To_ICxx.System_Faults[474]
		OR Out_To_ICxx.System_Faults[656]
		OR Out_To_ICxx.System_Faults[686]
		OR Out_To_ICxx.System_Faults[716];
	(*R27*)
	Out_To_ICxx.Rxx_UI_FaultPrompts.27:=
		Out_To_ICxx.System_Faults[481]
		OR Out_To_ICxx.System_Faults[482]
		OR Out_To_ICxx.System_Faults[483]
		OR Out_To_ICxx.System_Faults[484]
		OR Out_To_ICxx.System_Faults[657]
		OR Out_To_ICxx.System_Faults[687]
		OR Out_To_ICxx.System_Faults[717];
	(*R28*)
	Out_To_ICxx.Rxx_UI_FaultPrompts.28:=
		Out_To_ICxx.System_Faults[491]
		OR Out_To_ICxx.System_Faults[492]
		OR Out_To_ICxx.System_Faults[493]
		OR Out_To_ICxx.System_Faults[494]
		OR Out_To_ICxx.System_Faults[658]
		OR Out_To_ICxx.System_Faults[688]
		OR Out_To_ICxx.System_Faults[718];
	(*R29*)
	Out_To_ICxx.Rxx_UI_FaultPrompts.29:=
		Out_To_ICxx.System_Faults[501]
		OR Out_To_ICxx.System_Faults[502]
		OR Out_To_ICxx.System_Faults[503]
		OR Out_To_ICxx.System_Faults[504]
		OR Out_To_ICxx.System_Faults[659]
		OR Out_To_ICxx.System_Faults[689]
		OR Out_To_ICxx.System_Faults[719];
	(*R30*)
	Out_To_ICxx.Rxx_UI_FaultPrompts.30:=
		Out_To_ICxx.System_Faults[511]
		OR Out_To_ICxx.System_Faults[512]
		OR Out_To_ICxx.System_Faults[513]
		OR Out_To_ICxx.System_Faults[514]
		OR Out_To_ICxx.System_Faults[660]
		OR Out_To_ICxx.System_Faults[690]
		OR Out_To_ICxx.System_Faults[720];

	(*R1 - TSAFE ONLY*)
	Out_To_ICxx.Rxx_UI_FaultPrompts_2.1:=
		Out_To_ICxx.System_Faults[221]
		OR Out_To_ICxx.System_Faults[222]
		OR Out_To_ICxx.System_Faults[223]
		OR Out_To_ICxx.System_Faults[224];
	(*R2 - TSAFE ONLY*)
	Out_To_ICxx.Rxx_UI_FaultPrompts_2.2:=
		Out_To_ICxx.System_Faults[231]
		OR Out_To_ICxx.System_Faults[232]
		OR Out_To_ICxx.System_Faults[233]
		OR Out_To_ICxx.System_Faults[234];
	(*R3 - TSAFE ONLY*)
	Out_To_ICxx.Rxx_UI_FaultPrompts_2.3:=
		Out_To_ICxx.System_Faults[241]
		OR Out_To_ICxx.System_Faults[242]
		OR Out_To_ICxx.System_Faults[243]
		OR Out_To_ICxx.System_Faults[244];
	(*R4 - TSAFE ONLY*)
	Out_To_ICxx.Rxx_UI_FaultPrompts_2.4:=
		Out_To_ICxx.System_Faults[251]
		OR Out_To_ICxx.System_Faults[252]
		OR Out_To_ICxx.System_Faults[253]
		OR Out_To_ICxx.System_Faults[254];
	(*R5 - TSAFE ONLY*)
	Out_To_ICxx.Rxx_UI_FaultPrompts_2.5:=
		Out_To_ICxx.System_Faults[261]
		OR Out_To_ICxx.System_Faults[262]
		OR Out_To_ICxx.System_Faults[263]
		OR Out_To_ICxx.System_Faults[264];
	(*R6 - TSAFE ONLY*)
	Out_To_ICxx.Rxx_UI_FaultPrompts_2.6:=
		Out_To_ICxx.System_Faults[271]
		OR Out_To_ICxx.System_Faults[272]
		OR Out_To_ICxx.System_Faults[273]
		OR Out_To_ICxx.System_Faults[274];
	(*R7 - TSAFE ONLY*)
	Out_To_ICxx.Rxx_UI_FaultPrompts_2.7:=
		Out_To_ICxx.System_Faults[281]
		OR Out_To_ICxx.System_Faults[282]
		OR Out_To_ICxx.System_Faults[283]
		OR Out_To_ICxx.System_Faults[284];
	(*R8 - TSAFE ONLY*)
	Out_To_ICxx.Rxx_UI_FaultPrompts_2.8:=
		Out_To_ICxx.System_Faults[291]
		OR Out_To_ICxx.System_Faults[292]
		OR Out_To_ICxx.System_Faults[293]
		OR Out_To_ICxx.System_Faults[294];
	(*R9 - TSAFE ONLY*)
	Out_To_ICxx.Rxx_UI_FaultPrompts_2.9:=
		Out_To_ICxx.System_Faults[301]
		OR Out_To_ICxx.System_Faults[302]
		OR Out_To_ICxx.System_Faults[303]
		OR Out_To_ICxx.System_Faults[304];
	(*R10 - TSAFE ONLY*)
	Out_To_ICxx.Rxx_UI_FaultPrompts_2.10:=
		Out_To_ICxx.System_Faults[311]
		OR Out_To_ICxx.System_Faults[312]
		OR Out_To_ICxx.System_Faults[313]
		OR Out_To_ICxx.System_Faults[314];
	(*R11 - TSAFE ONLY*)
	Out_To_ICxx.Rxx_UI_FaultPrompts_2.11:=
		Out_To_ICxx.System_Faults[321]
		OR Out_To_ICxx.System_Faults[322]
		OR Out_To_ICxx.System_Faults[323]
		OR Out_To_ICxx.System_Faults[324];
	(*R12 - TSAFE ONLY*)
	Out_To_ICxx.Rxx_UI_FaultPrompts_2.12:=
		Out_To_ICxx.System_Faults[331]
		OR Out_To_ICxx.System_Faults[332]
		OR Out_To_ICxx.System_Faults[333]
		OR Out_To_ICxx.System_Faults[334];
	(*R13 - TSAFE ONLY*)
	Out_To_ICxx.Rxx_UI_FaultPrompts_2.13:=
		Out_To_ICxx.System_Faults[341]
		OR Out_To_ICxx.System_Faults[342]
		OR Out_To_ICxx.System_Faults[343]
		OR Out_To_ICxx.System_Faults[344];
	(*R14 - TSAFE ONLY*)
	Out_To_ICxx.Rxx_UI_FaultPrompts_2.14:=
		Out_To_ICxx.System_Faults[351]
		OR Out_To_ICxx.System_Faults[352]
		OR Out_To_ICxx.System_Faults[353]
		OR Out_To_ICxx.System_Faults[354];
	(*R15 - TSAFE ONLY*)
	Out_To_ICxx.Rxx_UI_FaultPrompts_2.15:=
		Out_To_ICxx.System_Faults[361]
		OR Out_To_ICxx.System_Faults[362]
		OR Out_To_ICxx.System_Faults[363]
		OR Out_To_ICxx.System_Faults[364];
	(*R16 - TSAFE ONLY*)
	Out_To_ICxx.Rxx_UI_FaultPrompts_2.16:=
		Out_To_ICxx.System_Faults[371]
		OR Out_To_ICxx.System_Faults[372]
		OR Out_To_ICxx.System_Faults[373]
		OR Out_To_ICxx.System_Faults[374];
	(*R17 - TSAFE ONLY*)
	Out_To_ICxx.Rxx_UI_FaultPrompts_2.17:=
		Out_To_ICxx.System_Faults[381]
		OR Out_To_ICxx.System_Faults[382]
		OR Out_To_ICxx.System_Faults[383]
		OR Out_To_ICxx.System_Faults[384];
	(*R18 - TSAFE ONLY*)
	Out_To_ICxx.Rxx_UI_FaultPrompts_2.18:=
		Out_To_ICxx.System_Faults[391]
		OR Out_To_ICxx.System_Faults[392]
		OR Out_To_ICxx.System_Faults[393]
		OR Out_To_ICxx.System_Faults[394];
	(*R19 - TSAFE ONLY*)
	Out_To_ICxx.Rxx_UI_FaultPrompts_2.19:=
		Out_To_ICxx.System_Faults[401]
		OR Out_To_ICxx.System_Faults[402]
		OR Out_To_ICxx.System_Faults[403]
		OR Out_To_ICxx.System_Faults[404];
	(*R20 - TSAFE ONLY*)
	Out_To_ICxx.Rxx_UI_FaultPrompts_2.20:=
		Out_To_ICxx.System_Faults[411]
		OR Out_To_ICxx.System_Faults[412]
		OR Out_To_ICxx.System_Faults[413]
		OR Out_To_ICxx.System_Faults[414];
	(*R21 - TSAFE ONLY*)
	Out_To_ICxx.Rxx_UI_FaultPrompts_2.21:=
		Out_To_ICxx.System_Faults[421]
		OR Out_To_ICxx.System_Faults[422]
		OR Out_To_ICxx.System_Faults[423]
		OR Out_To_ICxx.System_Faults[424];
	(*R22 - TSAFE ONLY*)
	Out_To_ICxx.Rxx_UI_FaultPrompts_2.22:=
		Out_To_ICxx.System_Faults[431]
		OR Out_To_ICxx.System_Faults[432]
		OR Out_To_ICxx.System_Faults[433]
		OR Out_To_ICxx.System_Faults[434];
	(*R23 - TSAFE ONLY*)
	Out_To_ICxx.Rxx_UI_FaultPrompts_2.23:=
		Out_To_ICxx.System_Faults[441]
		OR Out_To_ICxx.System_Faults[442]
		OR Out_To_ICxx.System_Faults[443]
		OR Out_To_ICxx.System_Faults[444];
	(*R24 - TSAFE ONLY*)
	Out_To_ICxx.Rxx_UI_FaultPrompts_2.24:=
		Out_To_ICxx.System_Faults[451]
		OR Out_To_ICxx.System_Faults[452]
		OR Out_To_ICxx.System_Faults[453]
		OR Out_To_ICxx.System_Faults[454];
	(*R25 - TSAFE ONLY*)
	Out_To_ICxx.Rxx_UI_FaultPrompts_2.25:=
		Out_To_ICxx.System_Faults[461]
		OR Out_To_ICxx.System_Faults[462]
		OR Out_To_ICxx.System_Faults[463]
		OR Out_To_ICxx.System_Faults[464];
	(*R26 - TSAFE ONLY*)
	Out_To_ICxx.Rxx_UI_FaultPrompts_2.26:=
		Out_To_ICxx.System_Faults[471]
		OR Out_To_ICxx.System_Faults[472]
		OR Out_To_ICxx.System_Faults[473]
		OR Out_To_ICxx.System_Faults[474];
	(*R27 - TSAFE ONLY*)
	Out_To_ICxx.Rxx_UI_FaultPrompts_2.27:=
		Out_To_ICxx.System_Faults[481]
		OR Out_To_ICxx.System_Faults[482]
		OR Out_To_ICxx.System_Faults[483]
		OR Out_To_ICxx.System_Faults[484];
	(*R28 - TSAFE ONLY*)
	Out_To_ICxx.Rxx_UI_FaultPrompts_2.28:=
		Out_To_ICxx.System_Faults[491]
		OR Out_To_ICxx.System_Faults[492]
		OR Out_To_ICxx.System_Faults[493]
		OR Out_To_ICxx.System_Faults[494];
	(*R29 - TSAFE ONLY*)
	Out_To_ICxx.Rxx_UI_FaultPrompts_2.29:=
		Out_To_ICxx.System_Faults[501]
		OR Out_To_ICxx.System_Faults[502]
		OR Out_To_ICxx.System_Faults[503]
		OR Out_To_ICxx.System_Faults[504];
	(*R30 - TSAFE ONLY*)
	Out_To_ICxx.Rxx_UI_FaultPrompts_2.30:=
		Out_To_ICxx.System_Faults[511]
		OR Out_To_ICxx.System_Faults[512]
		OR Out_To_ICxx.System_Faults[513]
		OR Out_To_ICxx.System_Faults[514];

		
	(*PD01*)
	Out_To_ICxx.ISxx_UI_FaultPrompts.1:=
		Out_To_ICxx.System_Faults[110]
		OR Out_To_ICxx.System_Faults[111]
		OR Out_To_ICxx.System_Faults[112]
		OR Out_To_ICxx.System_Faults[113]
		OR Out_To_ICxx.System_Faults[581]
		OR Out_To_ICxx.System_Faults[752];
		
	(*PD01 - TSAFE ONLY*)
	Out_To_ICxx.ISxx_UI_FaultPrompts.11:=
		Out_To_ICxx.System_Faults[110]
		OR Out_To_ICxx.System_Faults[111]
		OR Out_To_ICxx.System_Faults[112]
		OR Out_To_ICxx.System_Faults[113];

	(*ST01*)
	Out_To_ICxx.STxx_UI_FaultPrompts.1:=
		Out_To_ICxx.System_Faults[131]
		OR Out_To_ICxx.System_Faults[1465];
	(*ST02*)
	Out_To_ICxx.STxx_UI_FaultPrompts.2:=
		Out_To_ICxx.System_Faults[133]
		OR Out_To_ICxx.System_Faults[1466];
	(*ST03*)
	Out_To_ICxx.STxx_UI_FaultPrompts.3:=
		Out_To_ICxx.System_Faults[135]
		OR Out_To_ICxx.System_Faults[1467];
	(*ST04*)
	Out_To_ICxx.STxx_UI_FaultPrompts.4:=
		Out_To_ICxx.System_Faults[137]
		OR Out_To_ICxx.System_Faults[1468];

	(*ST01 - TSAFE ONLY*)
	Out_To_ICxx.STxx_UI_FaultPrompts.11:=
		Out_To_ICxx.System_Faults[131];
	(*ST02 - TSAFE ONLY*)
	Out_To_ICxx.STxx_UI_FaultPrompts.12:=
		Out_To_ICxx.System_Faults[133];
	(*ST03 - TSAFE ONLY*)
	Out_To_ICxx.STxx_UI_FaultPrompts.13:=
		Out_To_ICxx.System_Faults[135];
	(*ST04 - TSAFE ONLY*)
	Out_To_ICxx.STxx_UI_FaultPrompts.14:=
		Out_To_ICxx.System_Faults[137];

	(*MD01*)
	Out_To_ICxx.MDxx_UI_FaultPrompts.1:=
		Out_To_ICxx.System_Faults[551]
		OR Out_To_ICxx.System_Faults[571]
		OR Out_To_ICxx.System_Faults[1491];
	(*MD02*)
	Out_To_ICxx.MDxx_UI_FaultPrompts.2:=
		Out_To_ICxx.System_Faults[552]
		OR Out_To_ICxx.System_Faults[572]
		OR Out_To_ICxx.System_Faults[1492];
	(*MD03*)
	Out_To_ICxx.MDxx_UI_FaultPrompts.3:=
		Out_To_ICxx.System_Faults[553]
		OR Out_To_ICxx.System_Faults[573]
		OR Out_To_ICxx.System_Faults[1493];
	(*MD04*)
	Out_To_ICxx.MDxx_UI_FaultPrompts.4:=
		Out_To_ICxx.System_Faults[554]
		OR Out_To_ICxx.System_Faults[574]
		OR Out_To_ICxx.System_Faults[1494];
	(*MD05*)
	Out_To_ICxx.MDxx_UI_FaultPrompts.5:=
		Out_To_ICxx.System_Faults[555]
		OR Out_To_ICxx.System_Faults[575]
		OR Out_To_ICxx.System_Faults[1495];

	(*MD01 - TSAFE ONLY*)
	Out_To_ICxx.MDxx_UI_FaultPrompts.11:=
		Out_To_ICxx.System_Faults[551];
	(*MD02 - TSAFE ONLY*)
	Out_To_ICxx.MDxx_UI_FaultPrompts.12:=
		Out_To_ICxx.System_Faults[552];
	(*MD03 - TSAFE ONLY*)
	Out_To_ICxx.MDxx_UI_FaultPrompts.13:=
		Out_To_ICxx.System_Faults[553];
	(*MD04 - TSAFE ONLY*)
	Out_To_ICxx.MDxx_UI_FaultPrompts.14:=
		Out_To_ICxx.System_Faults[554];
	(*MD05 - TSAFE ONLY*)
	Out_To_ICxx.MDxx_UI_FaultPrompts.15:=
		Out_To_ICxx.System_Faults[555];


	(*SL01*)
	Out_To_ICxx.SLxx_UI_FaultPrompts.1:=
		Out_To_ICxx.System_Faults[1475];
	(*SL02*)
	Out_To_ICxx.SLxx_UI_FaultPrompts.2:=
		Out_To_ICxx.System_Faults[1476];
	(*SL03*)
	Out_To_ICxx.SLxx_UI_FaultPrompts.3:=
		Out_To_ICxx.System_Faults[1477];
	(*SL04*)
	Out_To_ICxx.SLxx_UI_FaultPrompts.4:=
		Out_To_ICxx.System_Faults[1478];
	(*SL05*)
	Out_To_ICxx.SLxx_UI_FaultPrompts.5:=
		Out_To_ICxx.System_Faults[1479];
	(*SL06*)
	Out_To_ICxx.SLxx_UI_FaultPrompts.6:=
		Out_To_ICxx.System_Faults[1480];
	(*SL07*)
	Out_To_ICxx.SLxx_UI_FaultPrompts.7:=
		Out_To_ICxx.System_Faults[1481];
	(*SL08*)
	Out_To_ICxx.SLxx_UI_FaultPrompts.8:=
		Out_To_ICxx.System_Faults[1482];
	(*SL09*)
	Out_To_ICxx.SLxx_UI_FaultPrompts.9:=
		Out_To_ICxx.System_Faults[1483];

	(*SS01*)
	Out_To_ICxx.MISCxx_UI_FaultPrompts.1:=
		Out_To_ICxx.System_Faults[584];
	(*SS02*)
	Out_To_ICxx.MISCxx_UI_FaultPrompts.2:=
		Out_To_ICxx.System_Faults[585];
	(*SS03*)
	Out_To_ICxx.MISCxx_UI_FaultPrompts.3:=
		Out_To_ICxx.System_Faults[586];

	(*ESW01*)
	Out_To_ICxx.MISCxx_UI_FaultPrompts.11:=
		Out_To_ICxx.System_Faults[587];
	(*ESW02*)
	Out_To_ICxx.MISCxx_UI_FaultPrompts.12:=
		Out_To_ICxx.System_Faults[588];
	(*ESW03*)
	Out_To_ICxx.MISCxx_UI_FaultPrompts.13:=
		Out_To_ICxx.System_Faults[589];
	(*ESW04*)
	Out_To_ICxx.MISCxx_UI_FaultPrompts.14:=
		Out_To_ICxx.System_Faults[590];


	
	(*NOTE, laser (LSRxx) fault prompts were never created when laser component was created*)
	(*the below are new placeholder added during TcUI migration, blt*)	
	(*LSR01*)
	Out_To_ICxx.MISCxx_UI_FaultPrompts.21:=
		FALSE;
	(*LSR02*)
	Out_To_ICxx.MISCxx_UI_FaultPrompts.22:=
		FALSE;
	(*LSR03*)
	Out_To_ICxx.MISCxx_UI_FaultPrompts.23:=
		FALSE;
	(*LSR04*)
	Out_To_ICxx.MISCxx_UI_FaultPrompts.24:=
		FALSE;
	(*LSR05*)
	Out_To_ICxx.MISCxx_UI_FaultPrompts.25:=
		FALSE;
	(*LSR06*)
	Out_To_ICxx.MISCxx_UI_FaultPrompts.26:=
		FALSE;
	(*LSR07*)
	Out_To_ICxx.MISCxx_UI_FaultPrompts.27:=
		FALSE;
	(*LSR08*)
	Out_To_ICxx.MISCxx_UI_FaultPrompts.28:=
		FALSE;
	(*LSR09*)
	Out_To_ICxx.MISCxx_UI_FaultPrompts.29:=
		FALSE;
		

	(*SD01*)
	Out_To_ICxx.SDxx_UI_FaultPrompts.1:=
		Out_To_ICxx.System_Faults[521]
		OR Out_To_ICxx.System_Faults[721]
		OR Out_To_ICxx.System_Faults[951]
		OR Out_To_ICxx.System_Faults[1531]
		OR Out_To_ICxx.System_Faults[1561];
	(*SD02*)
	Out_To_ICxx.SDxx_UI_FaultPrompts.2:=
		Out_To_ICxx.System_Faults[522]
		OR Out_To_ICxx.System_Faults[722]
		OR Out_To_ICxx.System_Faults[952]
		OR Out_To_ICxx.System_Faults[1532]
		OR Out_To_ICxx.System_Faults[1562];
	(*SD03*)
	Out_To_ICxx.SDxx_UI_FaultPrompts.3:=
		Out_To_ICxx.System_Faults[523]
		OR Out_To_ICxx.System_Faults[723]
		OR Out_To_ICxx.System_Faults[953]
		OR Out_To_ICxx.System_Faults[1533]
		OR Out_To_ICxx.System_Faults[1563];
	(*SD04*)
	Out_To_ICxx.SDxx_UI_FaultPrompts.4:=
		Out_To_ICxx.System_Faults[524]
		OR Out_To_ICxx.System_Faults[724]
		OR Out_To_ICxx.System_Faults[954]
		OR Out_To_ICxx.System_Faults[1534]
		OR Out_To_ICxx.System_Faults[1564];
	(*SD05*)
	Out_To_ICxx.SDxx_UI_FaultPrompts.5:=
		Out_To_ICxx.System_Faults[525]
		OR Out_To_ICxx.System_Faults[725]
		OR Out_To_ICxx.System_Faults[955]
		OR Out_To_ICxx.System_Faults[1535]
		OR Out_To_ICxx.System_Faults[1565];
	(*SD06*)
	Out_To_ICxx.SDxx_UI_FaultPrompts.6:=
		Out_To_ICxx.System_Faults[526]
		OR Out_To_ICxx.System_Faults[726]
		OR Out_To_ICxx.System_Faults[956]
		OR Out_To_ICxx.System_Faults[1536]
		OR Out_To_ICxx.System_Faults[1566];
	(*SD07*)
	Out_To_ICxx.SDxx_UI_FaultPrompts.7:=
		Out_To_ICxx.System_Faults[527]
		OR Out_To_ICxx.System_Faults[727]
		OR Out_To_ICxx.System_Faults[957]
		OR Out_To_ICxx.System_Faults[1537]
		OR Out_To_ICxx.System_Faults[1567];
	(*SD08*)
	Out_To_ICxx.SDxx_UI_FaultPrompts.8:=
		Out_To_ICxx.System_Faults[528]
		OR Out_To_ICxx.System_Faults[728]
		OR Out_To_ICxx.System_Faults[958]
		OR Out_To_ICxx.System_Faults[1538]
		OR Out_To_ICxx.System_Faults[1568];
	(*SD09*)
	Out_To_ICxx.SDxx_UI_FaultPrompts.9:=
		Out_To_ICxx.System_Faults[529]
		OR Out_To_ICxx.System_Faults[729]
		OR Out_To_ICxx.System_Faults[959]
		OR Out_To_ICxx.System_Faults[1539]
		OR Out_To_ICxx.System_Faults[1569];
	(*SD10*)
	Out_To_ICxx.SDxx_UI_FaultPrompts.10:=
		Out_To_ICxx.System_Faults[530]
		OR Out_To_ICxx.System_Faults[730]
		OR Out_To_ICxx.System_Faults[960]
		OR Out_To_ICxx.System_Faults[1540]
		OR Out_To_ICxx.System_Faults[1570];
	(*SD11*)
	Out_To_ICxx.SDxx_UI_FaultPrompts.11:=
		Out_To_ICxx.System_Faults[531]
		OR Out_To_ICxx.System_Faults[731]
		OR Out_To_ICxx.System_Faults[961]
		OR Out_To_ICxx.System_Faults[1541]
		OR Out_To_ICxx.System_Faults[1571];
	(*SD12*)
	Out_To_ICxx.SDxx_UI_FaultPrompts.12:=
		Out_To_ICxx.System_Faults[532]
		OR Out_To_ICxx.System_Faults[732]
		OR Out_To_ICxx.System_Faults[962]
		OR Out_To_ICxx.System_Faults[1542]
		OR Out_To_ICxx.System_Faults[1572];
	(*SD13*)
	Out_To_ICxx.SDxx_UI_FaultPrompts.13:=
		Out_To_ICxx.System_Faults[533]
		OR Out_To_ICxx.System_Faults[733]
		OR Out_To_ICxx.System_Faults[963]
		OR Out_To_ICxx.System_Faults[1543]
		OR Out_To_ICxx.System_Faults[1573];
	(*SD14*)
	Out_To_ICxx.SDxx_UI_FaultPrompts.14:=
		Out_To_ICxx.System_Faults[534]
		OR Out_To_ICxx.System_Faults[734]
		OR Out_To_ICxx.System_Faults[964]
		OR Out_To_ICxx.System_Faults[1544]
		OR Out_To_ICxx.System_Faults[1574];
	(*SD15*)
	Out_To_ICxx.SDxx_UI_FaultPrompts.15:=
		Out_To_ICxx.System_Faults[535]
		OR Out_To_ICxx.System_Faults[735]
		OR Out_To_ICxx.System_Faults[965]
		OR Out_To_ICxx.System_Faults[1545]
		OR Out_To_ICxx.System_Faults[1575];
	(*SD16*)
	Out_To_ICxx.SDxx_UI_FaultPrompts.16:=
		Out_To_ICxx.System_Faults[536]
		OR Out_To_ICxx.System_Faults[736]
		OR Out_To_ICxx.System_Faults[966]
		OR Out_To_ICxx.System_Faults[1546]
		OR Out_To_ICxx.System_Faults[1576];
	(*SD17*)
	Out_To_ICxx.SDxx_UI_FaultPrompts.17:=
		Out_To_ICxx.System_Faults[537]
		OR Out_To_ICxx.System_Faults[737]
		OR Out_To_ICxx.System_Faults[967]
		OR Out_To_ICxx.System_Faults[1547]
		OR Out_To_ICxx.System_Faults[1577];
	(*SD18*)
	Out_To_ICxx.SDxx_UI_FaultPrompts.18:=
		Out_To_ICxx.System_Faults[538]
		OR Out_To_ICxx.System_Faults[738]
		OR Out_To_ICxx.System_Faults[968]
		OR Out_To_ICxx.System_Faults[1548]
		OR Out_To_ICxx.System_Faults[1578];
	(*SD19*)
	Out_To_ICxx.SDxx_UI_FaultPrompts.19:=
		Out_To_ICxx.System_Faults[539]
		OR Out_To_ICxx.System_Faults[739]
		OR Out_To_ICxx.System_Faults[969]
		OR Out_To_ICxx.System_Faults[1549]
		OR Out_To_ICxx.System_Faults[1579];
	(*SD20*)
	Out_To_ICxx.SDxx_UI_FaultPrompts.20:=
		Out_To_ICxx.System_Faults[540]
		OR Out_To_ICxx.System_Faults[740]
		OR Out_To_ICxx.System_Faults[970]
		OR Out_To_ICxx.System_Faults[1550]
		OR Out_To_ICxx.System_Faults[1580];
	(*SD21*)
	Out_To_ICxx.SDxx_UI_FaultPrompts.21:=
		Out_To_ICxx.System_Faults[541]
		OR Out_To_ICxx.System_Faults[741]
		OR Out_To_ICxx.System_Faults[971]
		OR Out_To_ICxx.System_Faults[1551]
		OR Out_To_ICxx.System_Faults[1581];
	(*SD22*)
	Out_To_ICxx.SDxx_UI_FaultPrompts.22:=
		Out_To_ICxx.System_Faults[542]
		OR Out_To_ICxx.System_Faults[742]
		OR Out_To_ICxx.System_Faults[972]
		OR Out_To_ICxx.System_Faults[1552]
		OR Out_To_ICxx.System_Faults[1582];
	(*SD23*)
	Out_To_ICxx.SDxx_UI_FaultPrompts.23:=
		Out_To_ICxx.System_Faults[543]
		OR Out_To_ICxx.System_Faults[743]
		OR Out_To_ICxx.System_Faults[973]
		OR Out_To_ICxx.System_Faults[1553]
		OR Out_To_ICxx.System_Faults[1583];
	(*SD24*)
	Out_To_ICxx.SDxx_UI_FaultPrompts.24:=
		Out_To_ICxx.System_Faults[544]
		OR Out_To_ICxx.System_Faults[744]
		OR Out_To_ICxx.System_Faults[974]
		OR Out_To_ICxx.System_Faults[1554]
		OR Out_To_ICxx.System_Faults[1584];
	(*SD25*)
	Out_To_ICxx.SDxx_UI_FaultPrompts.25:=
		Out_To_ICxx.System_Faults[545]
		OR Out_To_ICxx.System_Faults[745]
		OR Out_To_ICxx.System_Faults[975]
		OR Out_To_ICxx.System_Faults[1555]
		OR Out_To_ICxx.System_Faults[1585];
	(*SD26*)
	Out_To_ICxx.SDxx_UI_FaultPrompts.26:=
		Out_To_ICxx.System_Faults[546]
		OR Out_To_ICxx.System_Faults[746]
		OR Out_To_ICxx.System_Faults[976]
		OR Out_To_ICxx.System_Faults[1556]
		OR Out_To_ICxx.System_Faults[1586];
	(*SD27*)
	Out_To_ICxx.SDxx_UI_FaultPrompts.27:=
		Out_To_ICxx.System_Faults[547]
		OR Out_To_ICxx.System_Faults[747]
		OR Out_To_ICxx.System_Faults[977]
		OR Out_To_ICxx.System_Faults[1557]
		OR Out_To_ICxx.System_Faults[1587];
	(*SD28*)
	Out_To_ICxx.SDxx_UI_FaultPrompts.28:=
		Out_To_ICxx.System_Faults[548]
		OR Out_To_ICxx.System_Faults[748]
		OR Out_To_ICxx.System_Faults[978]
		OR Out_To_ICxx.System_Faults[1558]
		OR Out_To_ICxx.System_Faults[1588];
	(*SD29*)
	Out_To_ICxx.SDxx_UI_FaultPrompts.29:=
		Out_To_ICxx.System_Faults[549]
		OR Out_To_ICxx.System_Faults[749]
		OR Out_To_ICxx.System_Faults[979]
		OR Out_To_ICxx.System_Faults[1559]
		OR Out_To_ICxx.System_Faults[1589];
	(*SD30*)
	Out_To_ICxx.SDxx_UI_FaultPrompts.30:=
		Out_To_ICxx.System_Faults[550]
		OR Out_To_ICxx.System_Faults[750]
		OR Out_To_ICxx.System_Faults[980]
		OR Out_To_ICxx.System_Faults[1560]
		OR Out_To_ICxx.System_Faults[1590];
	
	(*VFD01*)
	Out_To_ICxx.VFDxx_UI_FaultPrompts.1:=
		Out_To_ICxx.System_Faults[751]
		OR Out_To_ICxx.System_Faults[1501];
	(*VFD02*)
	Out_To_ICxx.VFDxx_UI_FaultPrompts.2:=
		Out_To_ICxx.System_Faults[752]
		OR Out_To_ICxx.System_Faults[1502];
	(*VFD03*)
	Out_To_ICxx.VFDxx_UI_FaultPrompts.3:=
		Out_To_ICxx.System_Faults[753]
		OR Out_To_ICxx.System_Faults[1503];
	(*VFD04*)
	Out_To_ICxx.VFDxx_UI_FaultPrompts.4:=
		Out_To_ICxx.System_Faults[754]
		OR Out_To_ICxx.System_Faults[1504];
	(*VFD05*)
	Out_To_ICxx.VFDxx_UI_FaultPrompts.5:=
		Out_To_ICxx.System_Faults[755]
		OR Out_To_ICxx.System_Faults[1505];


(*Gather Flags to Generate UI Prompting on Controls Button that links to Controls Menu*)
	General_Controls_Fault:=
		(*Configuration Fault*)
		Out_To_ICxx.System_Faults[0]
		(*Flags Generated Above*)
		OR (Out_To_ICxx.ICxx_UI_FaultPrompts<>0)
		OR (Out_To_ICxx.Rxx_UI_FaultPrompts<>0)
		OR (Out_To_ICxx.ISxx_UI_FaultPrompts<>0)
		OR (Out_To_ICxx.STxx_UI_FaultPrompts<>0)
		OR (Out_To_ICxx.SLxx_UI_FaultPrompts<>0)
		OR (Out_To_ICxx.NWxx_UI_FaultPrompts<>0)
		OR (Out_To_ICxx.MISCxx_UI_FaultPrompts<>0)
		OR (Out_To_ICxx.SDxx_UI_FaultPrompts<>0)
		OR (Out_To_ICxx.VFDxx_UI_FaultPrompts<>0)
		(*Internal Fixture Ecat Faults*)
		OR Out_To_ICxx.System_Faults[617]
		OR Out_To_ICxx.System_Faults[618]
		OR Out_To_ICxx.System_Faults[619]
		OR Out_To_ICxx.System_Faults[620]
		OR Out_To_ICxx.System_Faults[621]
		OR Out_To_ICxx.System_Faults[622]
		OR Out_To_ICxx.System_Faults[623]
		OR Out_To_ICxx.System_Faults[624]
		OR Out_To_ICxx.System_Faults[625]
		OR Out_To_ICxx.System_Faults[626]
		OR Out_To_ICxx.System_Faults[627]
		OR Out_To_ICxx.System_Faults[628];


(*!!!!!!!!!!!!!!!!!!!!!!!! Check Each Fault to Check Status and Develop Major and Minor Fault Flags As a Result If Fault Exsists !!!!!!!!!!!!!!!!!!!!!!!!!!!!!!!*)
(*!!!!!!!!!!!!!!!!!!!!!!!! Check Each Fault to Check Status and Develop Major and Minor Fault Flags As a Result If Fault Exsists !!!!!!!!!!!!!!!!!!!!!!!!!!!!!!!*)
(*!!!!!!!!!!!!!!!!!!!!!!!! Check Each Fault to Check Status and Develop Major and Minor Fault Flags As a Result If Fault Exsists !!!!!!!!!!!!!!!!!!!!!!!!!!!!!!!*)

(*Check Major Faults*)
FOR Loop_Index_Major:= 0 TO 990 DO
	IF (Loop_Index_Major>=0) AND (Loop_Index_Major<991) (*Ensure to check bounds to not run out of Array*)
		THEN System_Major_Fault:= Out_To_ICxx.System_Faults[Loop_Index_Major];
		IF System_Major_Fault
			THEN EXIT; (*Exit Loop upon first Fault Flagged*)
		END_IF;
	END_IF;
END_FOR;


(*Check Minor Faults*)
FOR Loop_Index_Minor:= 991 TO 1639 DO
	IF (Loop_Index_Minor>=991) AND (Loop_Index_Minor<1640) (*Ensure to check bounds to not run out of Array*)
		THEN System_Minor_Fault:= Out_To_ICxx.System_Faults[Loop_Index_Minor];
		IF System_Minor_Fault
			THEN EXIT; (*Exit Loop upon first Fault Flagged*)
		END_IF;
	END_IF;
END_FOR;

END_PROGRAM

(* stored: Version 1.1.0.1, ProductVersion 3.1.4024.12
   POU Faults: Id {e3e9c687-6dd1-49e4-a7be-79cb18cbd94e}, SpecialFunc None *)
